(* IEC 61131-3 sources: beebread/doc (part 3) *)

FUNCTION OSCAT_VERSION : DWORD
VAR_INPUT
	IN : BOOL;
END_VAR

IF in THEN
	OSCAT_VERSION := DATE_TO_DWORD(D#2024-07-16);
ELSE
	OSCAT_VERSION := 335;
END_IF;
END_FUNCTION

FUNCTION STATUS_TO_ESR : esr_data
VAR_INPUT
	status : BYTE;
	adress : STRING(10);
	DT_in : DT;
	TS : TIME;
END_VAR

IF status < 100 THEN
	status_to_ESR.typ := 1;
ELSIF status < 200 THEN
	status_to_ESR.typ := 2;
ELSE
	status_to_ESR.typ := 3;
END_IF;
status_to_ESR.adress:= adress;
status_to_ESR.DS := DT_in;
status_to_ESR.TS := TS;
status_to_ESR.data[0] := status;
END_FUNCTION

// Commented out for beedance: it reads or writes the bytes of a STRING through a pointer; a beedance reference (REF_TO) refers to a whole variable of its type.
// FUNCTION BIN_TO_BYTE : BYTE
// VAR_INPUT
// 	BIN : STRING(12);
// END_VAR
// VAR
// 	pt : REF_TO BYTE;
// 	i: INT;
// 	X: BYTE;
// 	stop: INT;
// END_VAR
//
// pt := REF(bin);
// stop := LEN(bin);
// FOR I := 1 TO stop DO
// 	x := pt^;
// 	(* calculate the value of the digit *)
// 	IF X = 48 THEN
// 		BIN_TO_BYTE := SHL(BIN_TO_BYTE,1);
// 	ELSIF X = 49 THEN
// 		BIN_TO_BYTE := SHL(BIN_TO_BYTE,1) OR 1;
// 	END_IF;
// 	pt := pt + 1;
// END_FOR;
// END_FUNCTION

// Commented out for beedance: it reads or writes the bytes of a STRING through a pointer; a beedance reference (REF_TO) refers to a whole variable of its type.
// FUNCTION BIN_TO_DWORD : DWORD
// VAR_INPUT
// 	BIN : STRING(40);
// END_VAR
// VAR
// 	pt : REF_TO BYTE;
// 	i: INT;
// 	X: BYTE;
// 	stop: INT;
// END_VAR
//
// pt := REF(bin);
// stop := LEN(bin);
// FOR I := 1 TO stop DO
// 	x := pt^;
// 	(* calculate the value of the digit *)
// 	IF X = 48 THEN
// 		BIN_TO_DWORD := SHL(BIN_TO_DWORD,1);
// 	ELSIF X = 49 THEN
// 		BIN_TO_DWORD := SHL(BIN_TO_DWORD,1) OR 1;
// 	END_IF;
// 	pt := pt + 1;
// END_FOR;
// END_FUNCTION

// Commented out for beedance: it computes with pointers as addresses (pt := pt + 1); beedance references (REF_TO) have no arithmetic.
// FUNCTION BYTE_TO_STRB : STRING(8)
// VAR_INPUT
// 	IN : BYTE;
// END_VAR
// VAR
// 	i: INT;
// 	pt : REF_TO BYTE;
// END_VAR
//
// (* determine pointer for the output *)
// pt := REF(BYTE_TO_STRB);
// (* determine and write the 8 output characters *)
// FOR i := 1 TO 8 DO
// 	pt^ := BOOL_TO_BYTE(in.7) + 48;
// 	in := SHL(in,1);
// 	pt := pt + 1;
// END_FOR;
//
// (* the output string still has to be terminated with 0 *)
// pt^ := 0;
// END_FUNCTION

// Commented out for beedance: it computes with pointers as addresses (pt := pt + 1); beedance references (REF_TO) have no arithmetic.
// FUNCTION BYTE_TO_STRH : STRING(2)
// VAR_INPUT
// 	IN : BYTE;
// END_VAR
// VAR
// 	temp : BYTE;
// 	PT : REF_TO BYTE;
// END_VAR
//
// (* read pointer to output string *)
// PT := REF(BYTE_TO_STRH);
// (* calculate high order hex value *)
// temp := SHR(in,4);
// (* convert value to hex character *)
// IF temp <= 9 THEN temp := temp + 48; ELSE temp := temp + 55; END_IF;
// (* write friat character to output string *)
// PT^ := temp;
// (* calculate low order hex value *)
// temp := in AND 2#00001111;
// IF temp <= 9 THEN temp := temp + 48; ELSE temp := temp + 55; END_IF;
// (* increment pointer and wirte low order character *)
// pt := pt + 1;
// pt^ := temp;
// (* set pointer at the end of the output string and close the string with 0 *)
// pt := pt + 1;
// pt^:= 0;
// END_FUNCTION

// Commented out for beedance: it computes with pointers as addresses (pt := pt + 1); beedance references (REF_TO) have no arithmetic.
// FUNCTION CAPITALIZE : STRING(STRING_LENGTH)
// VAR_INPUT
// 	str : STRING(STRING_LENGTH);
// END_VAR
// VAR
// 	PT : REF_TO BYTE;
// 	pos : INT;
// 	L : INT;
// 	first : BOOL := TRUE;
// END_VAR
//
// PT := REF(CAPITALIZE);
// CAPITALIZE := str;
// L := LEN(str);
// FOR pos := 1 TO l DO
// 	IF first THEN pt^ := TO_UPPER(pt^);	END_IF;
// 	(* remember in first if the next char needs to capitalized *)
// 	first := pt^= 32;
// 	PT := pt + 1;
// END_FOR;
// END_FUNCTION

// Commented out for beedance: it uses CODE, which is commented out.
// FUNCTION CHARCODE : BYTE
// VAR_INPUT
// 	STR : STRING(10);
// END_VAR
// VAR
// 	found: STRING(1);
// 	search : STRING(10);
// 	pos: INT;
// 	i: INT;
// END_VAR
//
// IF LEN(str) = 1 THEN
// 	CHARCODE := CODE(STR, 1);
// ELSIF str <> '' THEN
// 	(* construct search string *)
// 	search := CONCAT('&', str);
// 	search := CONCAT(search, ';');
// 	WHILE pos = 0 AND (i < 4) DO
// 		i := i + 1;
// 		pos := FIND(setup.CHARNAMES[i], search);
// 	END_WHILE;
// 	found := MID(setup.CHARNAMES[i], 1, pos - 1);
// 	CHARCODE := CODE(found, 1);
// END_IF;
// END_FUNCTION

// Commented out for beedance: it uses CHR_TO_STRING, which is commented out.
// FUNCTION CHARNAME : STRING(10)
// VAR_INPUT
// 	C : BYTE;
// END_VAR
// VAR
// 	pos: INT;
// 	i : INT;
// END_VAR
//
// IF C <> 0 THEN
// 	(* construct search string from code followed by $ sign, also clear charname string*)
// 	CHARNAME := CHR_TO_STRING(C);
// 	CHARNAME := CONCAT(CHARNAME,'&');
// 	CHARNAME := CONCAT(';', CHARNAME);
// 	WHILE pos = 0 AND (i < 4) DO
// 		i := i + 1;
// 		pos := FIND(setup.CHARNAMES[i], CHARNAME);
// 	END_WHILE;
// 	IF pos > 0 THEN
// 		CHARNAME := MID(setup.CHARNAMES[i], 10, pos + 3);
// 		(* search for end of name and truncate *)
// 		pos := FIND(CHARNAME, ';');
// 		CHARNAME := LEFT(CHARNAME,pos - 1);
// 	ELSE
// 		CHARNAME := CHR_TO_STRING(C);
// 	END_IF;
// ELSE
// 	CHARNAME := '';
// END_IF;
// END_FUNCTION

// Commented out for beedance: it computes with pointers as addresses (pt := pt + 1); beedance references (REF_TO) have no arithmetic.
// FUNCTION CHR_TO_STRING : STRING(1)
// VAR_INPUT
// 	C : BYTE;
// END_VAR
// VAR
// 	PT : REF_TO BYTE;
// END_VAR
//
// PT := REF(CHR_TO_STRING);
// PT^ := C;
// pt := pt + 1;
// pt^ := 0;
// END_FUNCTION

FUNCTION CLEAN : STRING(STRING_LENGTH)
VAR_INPUT
	IN : STRING(STRING_LENGTH);
	CX : STRING(80);
END_VAR
VAR
	pos: INT := 1;
	stop: INT;
END_VAR

(* copy input string *)
CLEAN := IN;
stop := LEN(in);
WHILE pos <= stop DO
	IF FIND(cx, MID(CLEAN, 1, pos)) > 0 THEN
		(* charcter found skip to next one *)
		pos := pos + 1;
	ELSE
		(* wrong chracter needs to be deleted *)
		CLEAN := DELETE(CLEAN, 1, pos);
		stop := stop - 1;	(* the string is one character shorter now *)
	END_IF;
END_WHILE;
END_FUNCTION

// Commented out for beedance: it computes with pointers as addresses (pt := pt + 1); beedance references (REF_TO) have no arithmetic.
// FUNCTION CODE : BYTE
// VAR_INPUT
// 	STR : STRING(STRING_LENGTH);
// 	POS : INT;
// END_VAR
// VAR
// 	PT : REF_TO BYTE;
// END_VAR
//
// IF pos < 1 OR pos > LEN(str) THEN
// 	CODE := 0;
// 	RETURN;
// ELSE
// 	PT := REF(STR) + INT_TO_DWORD(pos - 1);
// 	CODE := pt^;
// END_IF;
// END_FUNCTION

// Commented out for beedance: it reads or writes the bytes of a STRING through a pointer; a beedance reference (REF_TO) refers to a whole variable of its type.
// FUNCTION COUNT_CHAR : INT
// VAR_INPUT
// 	str : STRING(STRING_LENGTH);
// 	chr : BYTE;
// END_VAR
// VAR
// 	l: INT;
// 	pt : REF_TO BYTE;
// 	pos: INT;
// END_VAR
//
// PT := REF(str);
// l := LEN(str);
// COUNT_CHAR := 0;
// FOR pos := 1 TO l DO
// 	IF pt^ = CHR THEN COUNT_CHAR := COUNT_CHAR + 1; END_IF;
//     PT := PT + 1;
// END_FOR;
// END_FUNCTION

FUNCTION COUNT_SUBSTRING : INT
VAR_INPUT
   SEARCH : STRING;
   STR : STRING;
END_VAR
VAR
   pos : INT;
   size : INT;
END_VAR
VAR
	STR_work : STRING;
END_VAR
(* IEC 61131-3 does not let a POU assign to its inputs, so the body works on copies. *)
STR_work := STR;

COUNT_SUBSTRING := 0;
size := LEN(SEARCH);
REPEAT
   pos := FIND(STR_work,SEARCH);
   IF pos > 0 THEN
      STR_work := REPLACE(STR_work, '', size,pos);
      COUNT_SUBSTRING := COUNT_SUBSTRING + 1;
   END_IF;
UNTIL pos = 0
END_REPEAT;
END_FUNCTION

// Commented out for beedance: it reads or writes the bytes of a STRING through a pointer; a beedance reference (REF_TO) refers to a whole variable of its type.
// FUNCTION DEC_TO_BYTE : BYTE
// VAR_INPUT
// 	DEC : STRING(10);
// END_VAR
// VAR
// 	pt : REF_TO BYTE;
// 	i: INT;
// 	X: BYTE;
// 	stop: INT;
// END_VAR
//
// pt := REF(dec);
// stop := LEN(DEC);
// FOR I := 1 TO stop DO
// 	(* read the first character and subtract 48 to get value in decimal 0 = 48 *)
// 	x := pt^;
// 	(* calculate the value of the digit *)
// 	IF X > 47 AND x < 58 THEN
// 		DEC_TO_BYTE := DEC_TO_BYTE * 10 + X - 48;
// 	END_IF;
// 	pt := pt + 1;
// END_FOR;
// END_FUNCTION

// Commented out for beedance: it reads or writes the bytes of a STRING through a pointer; a beedance reference (REF_TO) refers to a whole variable of its type.
// FUNCTION DEC_TO_DWORD : DWORD
// VAR_INPUT
// 	DEC : STRING(20);
// END_VAR
// VAR
// 	pt : REF_TO BYTE;
// 	i: INT;
// 	X: BYTE;
// 	stop: INT;
// END_VAR
//
// pt := REF(dec);
// stop := LEN(dec);
// FOR I := 1 TO stop DO
// 	(* read the first character and subtract 48 to get value in decimal 0 = 48 *)
// 	x := pt^;
// 	(* calculate the value of the digit *)
// 	IF X > 47 AND x < 58 THEN
// 		DEC_TO_DWORD := DEC_TO_DWORD * 10 + X - 48;
// 	END_IF;
// 	pt := pt + 1;
// END_FOR;
// END_FUNCTION

// Commented out for beedance: it reads or writes the bytes of a STRING through a pointer; a beedance reference (REF_TO) refers to a whole variable of its type.
// FUNCTION DEC_TO_INT : INT
// VAR_INPUT
// 	DEC : STRING(10);
// END_VAR
// VAR
// 	pt : REF_TO BYTE;
// 	i: INT;
// 	X: BYTE;
// 	sign: BOOL;
// 	stop: INT;
// END_VAR
//
// pt := REF(dec);
// stop := LEN(dec);
// FOR I := 1 TO stop DO
// 	(* read the first character and subtract 48 to get value in decimal 0 = 48 *)
// 	x := pt^;
// 	(* calculate the value of the digit *)
// 	IF X > 47 AND x < 58 THEN
// 		DEC_TO_INT := DEC_TO_INT * 10 + X - 48;
// 	ELSIF X = 45 AND DEC_TO_INT = 0 THEN
// 		sign := TRUE;
// 	END_IF;
// 	pt := pt + 1;
// END_FOR;
// IF sign THEN DEC_TO_INT := -DEC_TO_INT; END_IF;
// END_FUNCTION

FUNCTION DEL_CHARS : STRING(STRING_LENGTH)
VAR_INPUT
	IN : STRING(STRING_LENGTH);
	CX : STRING(80);
END_VAR
VAR
	pos: INT := 1;
	stop: INT;
END_VAR

(* copy input string *)
DEL_CHARS := IN;
stop := LEN(in);
WHILE pos <= stop DO
	IF FIND(cx, MID(DEL_CHARS, 1, pos)) > 0 THEN
		(* wrong chracter needs to be deleted *)
		DEL_CHARS := DELETE(DEL_CHARS, 1, pos);
		stop := stop - 1;	(* the string is one character shorter now *)
	ELSE
		(* charcter not found skip to next one *)
		pos := pos + 1;
	END_IF;
END_WHILE;
END_FUNCTION

// Commented out for beedance: it uses CODE, which is commented out.
// FUNCTION DT_TO_STRF : STRING
// VAR_INPUT
// 	DTI : DT;
// 	MS : INT;
// 	FMT : STRING;
// 	LANG : INT;
// END_VAR
// VAR CONSTANT
// 	FILL : STRING(1) := '0';
// 	BLANK : STRING(1) := ' ';
// END_VAR
// VAR
// 	ly : INT;
// 	dx: DATE;
// 	fs: STRING(10);
// 	td: TOD;
// 	tmp : INT;
// 	pos : INT;
// 	f : INT;
// END_VAR
//
// IF LANG < 1 THEN ly := language.DEFAULT; ELSE ly := MIN(language.LMAX, LANG); END_IF;
//
// (* decode date and time information *)
// dx := DT_TO_DATE(DTI);
// td := DT_TO_TOD(DTI);
//
// (* parse the format string *)
// DT_TO_STRF := FMT;
// pos := FIND(DT_TO_STRF, '#');
// WHILE pos > 0 DO
// 	(* retrieve format identifier *)
// 	f := CODE(DT_TO_STRF, pos + 1);
// 	(* generate the return string according to the format character *)
// 	fs := '';
// 	CASE f OF
// 		65 : (* letter A retunrs the year in 4 digits *)
// 			fs := INT_TO_STRING(YEAR_OF_DATE(dx));
// 		66 : (* letter B returns the year in exactly 2 digits *)
// 			fs := RIGHT(INT_TO_STRING(YEAR_OF_DATE(dx)),2);
// 		67 : (* letter C returns the month with 1 or 2 digits *)
// 			fs := INT_TO_STRING(MONTH_OF_DATE(dx));
// 		68 : (* letter D returns the month with exactly 2 digits *)
// 			fs := INT_TO_STRING(MONTH_OF_DATE(dx));
// 			IF LEN(fs) < 2 THEN fs := CONCAT('0', fs); END_IF;
// 		69 : (* letter E returns the month with 3 characters *)
// 			fs := MONTH_TO_STRING(MONTH_OF_DATE(dx), ly, 3);
// 		70 : (* letter F returns the month with all characters *)
// 			fs := MONTH_TO_STRING(MONTH_OF_DATE(dx), ly, 0);
// 		71 : (* letter G returns the day with up to 2 digits *)
// 			fs := INT_TO_STRING(DAY_OF_MONTH(dx));
// 		72 : (* letter H returns the day of the month with exactly 2 digits *)
// 			fs := INT_TO_STRING(DAY_OF_MONTH(dx));
// 			IF LEN(fs) < 2 THEN fs := CONCAT(FILL, fs); END_IF;
// 		73 : (* letter I returns the weekday as the number 1..7 1 = monday *)
// 			fs := INT_TO_STRING(DAY_OF_WEEK(dx));
// 		74 : (* letter J returns the weekday in 2 character writing *)
// 			fs := WEEKDAY_TO_STRING(DAY_OF_WEEK(dx), ly, 2);
// 		75 : (* letter K returns the weekday with all characters *)
// 			fs := WEEKDAY_TO_STRING(DAY_OF_WEEK(dx), ly, 0);
// 		76 : (* letter L returns AM or PM for the given DateTime *)
// 			IF td >= TOD#12:00:00 THEN fs := 'PM'; ELSE fs := 'AM'; END_IF;
// 		77 : (* letter M returns the hour in 1 or 2 digit form 0..24h *)
// 			fs := INT_TO_STRING(HOUR(td));
// 		78 : (* letter N returns the hour in exactly 2 digit form 0..24h *)
// 			fs := INT_TO_STRING(HOUR(td));
// 			IF LEN(fs) < 2 THEN fs := CONCAT(FILL, fs); END_IF;
// 		79 : (* letter O returns the hour in 1 or 2 digit form 0..12h *)
// 			tmp := HOUR(td) MOD 12;
// 			IF tmp = 0 THEN tmp := 12; END_IF;
// 			fs := INT_TO_STRING(tmp);
// 		80 : (* letter P returns the hour in exactly 2 digit form 0..12h *)
// 			tmp := HOUR(td) MOD 12;
// 			IF tmp = 0 THEN tmp := 12; END_IF;
// 			fs := INT_TO_STRING(tmp);
// 			IF LEN(fs) < 2 THEN fs := CONCAT(FILL, fs); END_IF;
// 		81 : (* letter Q returns the minute of the hour in 1 or two digit form *)
// 			fs := INT_TO_STRING(MINUTE(td));
// 		82 : (* letter R returns the minute of the hour in exactly two digit form *)
// 			fs := INT_TO_STRING(MINUTE(td));
// 			IF LEN(fs) < 2 THEN fs := CONCAT(FILL, fs); END_IF;
// 		83 : (* letter S returns the second of the minute in 1 or two digit form *)
// 			fs := INT_TO_STRING(REAL_TO_INT(SECOND(td)));
// 		84 : (* letter T returns the second of the minute in exactly two digit form *)
// 			fs := INT_TO_STRING(REAL_TO_INT(SECOND(td)));
// 			IF LEN(fs) < 2 THEN fs := CONCAT(FILL, fs); END_IF;
// 		85 : (* letter U returns the milliseconds in 1 to 3 digits *)
// 			fs := INT_TO_STRING(MS);
// 		86 : (* letter V returns the milliseconds in exactly 3 digit form *)
// 			fs := INT_TO_STRING(MS);
// 			fs := CONCAT('00',fs);
// 			fs := RIGHT(fs, 3);
// 		87 : (* letter W returns the day of the month with exactly 2 digits first digit is filled with blank if necessary *)
// 			fs := INT_TO_STRING(DAY_OF_MONTH(dx));
// 			IF LEN(fs) < 2 THEN fs := CONCAT(BLANK, fs); END_IF;
// 		88 : (* letter X returns the month with exactly 2 digits first digit is filled with blank if necessary *)
// 			fs := INT_TO_STRING(MONTH_OF_DATE(dx));
// 			IF LEN(fs) < 2 THEN fs := CONCAT(BLANK, fs); END_IF;
// 		END_CASE;
// 	DT_TO_STRF := REPLACE(DT_TO_STRF, fs, 2, pos);
// 	pos := FIND(DT_TO_STRF, '#');
// END_WHILE;
// END_FUNCTION

// Commented out for beedance: it computes with pointers as addresses (pt := pt + 1); beedance references (REF_TO) have no arithmetic.
// FUNCTION DWORD_TO_STRB : STRING(32)
// VAR_INPUT
// 	IN : DWORD;
// END_VAR
// VAR
// 	pt : REF_TO BYTE;
// 	i: INT;
// END_VAR
//
// (* determine pointer for the output *)
// pt := REF(DWORD_TO_STRB);
// (* determine and write the 8 output characters *)
// FOR i := 1 TO 32 DO
// 	pt^:= BOOL_TO_BYTE(in.31) + 48;
// 	in := SHL(in,1);
// 	pt := pt + 1;
// END_FOR;
//
// (* the output string still has to be terminated with 0 *)
// pt^ := 0;
// END_FUNCTION

// Commented out for beedance: it uses FIX, which is commented out.
// FUNCTION DWORD_TO_STRF : STRING(20)
// VAR_INPUT
// 	IN : DWORD;
// 	N : INT;
// END_VAR
//
// (* limit N to max 20 characters *)
// (* convert dword to string first and cut to length N *)
// DWORD_TO_STRF := FIX(DWORD_TO_STRING(in),LIMIT(0,N,20),48,1);
// END_FUNCTION

// Commented out for beedance: it computes with pointers as addresses (pt := pt + 1); beedance references (REF_TO) have no arithmetic.
// FUNCTION DWORD_TO_STRH : STRING(8)
// VAR_INPUT
// 	IN : DWORD;
// END_VAR
// VAR
// 	i : INT;
// 	temp : BYTE;
// 	pt : REF_TO BYTE;
// END_VAR
//
// (* read output adress to pointer *)
// pt := REF(DWORD_TO_STRH) + 8;
// (* wirte the closing byte for the string *)
// pt^:= 0;
//
// (* write the 8 hex characters backwards *)
// FOR i := 1 TO 8 DO;
// 	(* decrement the pointer *)
// 	pt := pt - 1;
// 	(* read the lowest order hex value *)
// 	temp := DWORD_TO_BYTE(in AND 16#0000000F);
// 	(* convert value to hex character *)
// 	IF temp <= 9 THEN temp := temp + 48; ELSE temp := temp + 55; END_IF;
// 	(* write character to output string *)
// 	PT^ := temp;
// 	(* shift in for nect hex character *)
// 	in := SHR(in,4);
// END_FOR;
// END_FUNCTION

// Commented out for beedance: it uses UPPERCASE, which is commented out.
// FUNCTION EXEC : STRING(STRING_LENGTH)
// VAR_INPUT
// 	str : STRING(STRING_LENGTH);
// END_VAR
// VAR
// 	pos: INT;
// 	R1: REAL;
// 	R2: REAL;
// 	operator: STRING(10);
// END_VAR
//
// (* extract both numbers and operator *)
// EXEC := UPPERCASE(TRIM(str));
//
// pos := FINDB_NONUM(EXEC);
// IF pos > 1 THEN R1 := STRING_TO_REAL(LEFT(EXEC,pos-1)); END_IF;
// R2 := STRING_TO_REAL(RIGHT(EXEC,LEN(EXEC)-pos));
// EXEC := LEFT(EXEC,pos);
// pos := FINDB_NUM(EXEC);
// operator := RIGHT(EXEC,LEN(EXEC) - pos);
// IF operator = '' AND LEN(str) = 0 THEN
// 	EXEC := '';
// 	RETURN;
// ELSIF operator = '' THEN
// 	EXEC := str;
// 	RETURN;
// END_IF;
// IF operator = '^' THEN
// 	EXEC := REAL_TO_STRING(EXPT(R1, R2));
// ELSIF operator = 'SQRT' THEN
// 	EXEC := REAL_TO_STRING(SQRT(R2));
// ELSIF operator = 'SIN' THEN
// 	EXEC := REAL_TO_STRING(SIN(r2));
// ELSIF operator = 'COS' THEN
// 	EXEC := REAL_TO_STRING(COS(r2));
// ELSIF operator = 'TAN' THEN
// 	EXEC := REAL_TO_STRING(TAN(R2));
// ELSIF operator = '*' THEN
// 	EXEC := REAL_TO_STRING(R1 * R2);
// ELSIF operator = '/' THEN
// 	IF R2 <> 0 THEN EXEC := REAL_TO_STRING(R1 / R2); ELSE EXEC := 'ERROR'; END_IF;
// ELSIF operator = '+' THEN
// 	EXEC := REAL_TO_STRING(r1 + r2);
// ELSIF operator = '-' THEN
// 	EXEC := REAL_TO_STRING(r1 - r2);
// ELSE
// 	EXEC := 'ERROR';
// END_IF;
//
// IF EXEC = 'ERROR' THEN
// 	RETURN;
// (* some systems deliver integer instead of real *)
// ELSIF FIND(EXEC,'.') = 0 THEN
// 	EXEC := CONCAT(EXEC, '.0');
// (* some systems deliver n. instead of n.0 ! *)
// ELSIF RIGHT(EXEC,1) = '.' THEN
// 	EXEC := CONCAT(EXEC,'0');
// END_IF;
// END_FUNCTION

// Commented out for beedance: it uses CHR_TO_STRING, which is commented out.
// FUNCTION FILL : STRING(STRING_LENGTH)
// VAR_INPUT
// 	C : BYTE;
// 	L : INT;
// END_VAR
// VAR
// 	i: INT;
// 	sx: STRING(1);
// END_VAR
// VAR
// 	L_work : INT;
// END_VAR
// (* IEC 61131-3 does not let a POU assign to its inputs, so the body works on copies. *)
// L_work := L;
//
// Sx := CHR_TO_STRING(c);
// (* limit L to maximum 80 characters the length of a standard string *)
// L_work := LIMIT(0,L_work,STRING_LENGTH);
// (* create a string of characters to be connected to str *)
// FOR i := 1 TO 8 DO
// 	FILL := CONCAT(FILL,FILL);
// 	IF L_work.7 THEN FILL := CONCAT(FILL,Sx); END_IF;
// 	L_work := SHL(L_work,1);
// END_FOR;
// END_FUNCTION

// Commented out for beedance: it reads or writes the bytes of a STRING through a pointer; a beedance reference (REF_TO) refers to a whole variable of its type.
// FUNCTION FIND_CHAR : INT
// VAR_INPUT
// 	str : STRING(STRING_LENGTH);
// 	pos : INT;
// END_VAR
// VAR
// 	i: INT;
// 	pt : REF_TO ARRAY[1..255] OF BYTE;
// 	stop: INT;
// 	X: BYTE;
// END_VAR
//
// pt := REF(str);
// stop := LEN(str);
// FOR i := MAX(pos,1) TO stop DO;
// 	X := pt^[i];
// 	IF X > 31 AND ((setup.EXTENDED_ASCII AND X <> 127) OR (NOT setup.EXTENDED_ASCII AND X < 127)) THEN
// 		FIND_CHAR := i;
// 		RETURN;
// 	END_IF;
// END_FOR;
// FIND_CHAR := 0;
// END_FUNCTION

// Commented out for beedance: it reads or writes the bytes of a STRING through a pointer; a beedance reference (REF_TO) refers to a whole variable of its type.
// FUNCTION FIND_CTRL : INT
// VAR_INPUT
// 	str : STRING(STRING_LENGTH);
// 	pos : INT;
// END_VAR
// VAR
// 	i: INT;
// 	pt : REF_TO ARRAY[1..255] OF BYTE;
// 	stop: INT;
// 	x: BYTE;
// END_VAR
//
// pt := REF(str);
// stop := LEN(str);
// FOR i := MAX(pos,1) TO stop DO;
// 	x := PT^[I];
// 	IF x < 32 OR X = 127 THEN
// 		FIND_CTRL := i;
// 		RETURN;
// 	END_IF;
// END_FOR;
// FIND_CTRL := 0;
// END_FUNCTION

// Commented out for beedance: it reads or writes the bytes of a STRING through a pointer; a beedance reference (REF_TO) refers to a whole variable of its type.
// FUNCTION FIND_NONUM : INT
// VAR_INPUT
// 	str : STRING(STRING_LENGTH);
// 	pos : INT;
// END_VAR
// VAR
// 	i: INT;
// 	pt : REF_TO ARRAY[1..255] OF BYTE;
// 	end: INT;
// 	X: BYTE;
// END_VAR
//
// pt := REF(str);
// end := LEN(str);
// FOR i := MAX(pos,1) TO end DO;
// 	X := pt^[i];
// 	IF (X < 48 AND X <> 46) OR X > 57 THEN
// 		FIND_NONUM := i;
// 		RETURN;
// 	END_IF;
// END_FOR;
// FIND_NONUM := 0;
// END_FUNCTION

// Commented out for beedance: it reads or writes the bytes of a STRING through a pointer; a beedance reference (REF_TO) refers to a whole variable of its type.
// FUNCTION FIND_NUM : INT
// VAR_INPUT
// 	str : STRING(STRING_LENGTH);
// 	pos : INT;
// END_VAR
// VAR
// 	i : INT;
// 	pt : REF_TO ARRAY[1..255] OF BYTE;
// 	stop : INT;
// 	X: BYTE;
// END_VAR
//
// pt := REF(str);
// stop := LEN(str);
// FOR i := MAX(pos,1) TO stop DO;
// 	X := pt^[i];
// 	IF (X > 47 AND X < 58) OR X = 46 THEN
// 		FIND_NUM := i;
// 		RETURN;
// 	END_IF;
// END_FOR;
// FIND_NUM := 0;
// END_FUNCTION

FUNCTION FINDB : INT
VAR_INPUT
	str1 : STRING(STRING_LENGTH);
	str2 : STRING(STRING_LENGTH);
END_VAR
VAR
	pos: INT;
	length: INT;
END_VAR

length := LEN(str2);
FOR pos := LEN(str1) - length + 1 TO 1 BY -1 DO
	IF MID(str1,length,pos) = str2 THEN
		FindB := pos;
		RETURN;
	END_IF;
END_FOR;
FindB := 0;
END_FUNCTION

// Commented out for beedance: it computes with pointers as addresses (pt := pt + 1); beedance references (REF_TO) have no arithmetic.
// FUNCTION FINDB_NONUM : INT
// VAR_INPUT
// 	str : STRING(STRING_LENGTH);
// END_VAR
// VAR
// 	pos: INT;
// 	pt : REF_TO BYTE;
// END_VAR
//
// pt := REF(str) + LEN(str) - 1;
// FOR pos := LEN(str) TO 1 BY -1 DO;
// 	IF (PT^ < 48 AND PT^ <> 46) OR PT^ > 57 THEN
// 		FINDB_NONUM := pos;
// 		RETURN;
// 	END_IF;
// 	PT := PT - 1;
// END_FOR;
// FINDB_NONUM := 0;
// END_FUNCTION

// Commented out for beedance: it computes with pointers as addresses (pt := pt + 1); beedance references (REF_TO) have no arithmetic.
// FUNCTION FINDB_NUM : INT
// VAR_INPUT
// 	str : STRING(STRING_LENGTH);
// END_VAR
// VAR
// 	pos: INT;
// 	pt : REF_TO BYTE;
// END_VAR
//
// pt := REF(str) + LEN(str) - 1;
// FOR pos := LEN(str) TO 1 BY -1 DO;
// 	IF (PT^ > 47 AND PT^ < 58) OR PT^ = 46 THEN
// 		FINDB_NUM := pos;
// 		RETURN;
// 	END_IF;
// 	PT := PT - 1;
// END_FOR;
// FINDB_NUM := 0;
// END_FUNCTION

FUNCTION FINDP : INT
VAR_INPUT
	str : STRING(STRING_LENGTH);
	src : STRING(STRING_LENGTH);
	pos: INT;
END_VAR
VAR
	i: INT;
	ls: INT;
	lx: INT;
	stp: INT;
END_VAR

ls := LEN(str);
lx := LEN(src);
IF ls < lx OR lx = 0 THEN RETURN; END_IF;
stp := ls - lx + 1;
FOR i := MAX(pos,1) TO stp DO
	IF MID(str,lx,i) = src THEN
		FINDP := i;
		RETURN;
	END_IF;
END_FOR;
FINDP := 0;
END_FUNCTION

// Commented out for beedance: it uses FILL, which is commented out.
// FUNCTION FIX : STRING(STRING_LENGTH)
// VAR_INPUT
// 	str : STRING(STRING_LENGTH);
// 	L : INT;
// 	C : BYTE;
// 	M : INT;
// END_VAR
// VAR
// 	N : INT;
// 	SX: STRING(STRING_LENGTH);
// END_VAR
//
// (* make sure L does not exceed the limits of a string *)
// N := LIMIT(0,L,STRING_LENGTH) - LEN(str);
// IF N <= 0 THEN
// 	(* truncate the string at length N *)
// 	IF M = 1 THEN
// 		FIX := RIGHT(str,L);
// 	ELSE
// 		FIX := LEFT(str,L);
// 	END_IF;
// ELSIF M = 1 THEN
// 	(* connect fill characters at the beginning *)
// 	sx := FILL(C,N);
// 	FIX := CONCAT(sx,str);
// ELSIF M = 2 THEN
// 	(* center str beween fill characters *)
// 	(* for an uneven number of fill characters, there is one more at the end *)
// 	sx := FILL(C,SHR(N+1,1));
// 	FIX := CONCAT(str,sx);
// 	SX := LEFT(sx,SHR(N,1));
// 	FIX := CONCAT(sx,FIX);
// ELSE
// 	(* connect fill characters at the end *)
// 	SX := FILL(C,N);
// 	FIX := CONCAT(str,SX);
// END_IF;
// END_FUNCTION

// Commented out for beedance: it reads or writes the bytes of a STRING through a pointer; a beedance reference (REF_TO) refers to a whole variable of its type.
// FUNCTION FLOAT_TO_REAL : REAL
// VAR_INPUT
// 	FLT : STRING(20);
// END_VAR
// VAR
// 	pt : REF_TO ARRAY[1..20] OF BYTE;
// 	i: INT;
// 	X: BYTE;
// 	sign: INT := 1;
// 	stop: INT;
// 	tmp: DINT;
// 	d : INT;
// END_VAR
//
// pt := REF(FLT);
// stop := LEN(FLT);
//
// (* we first check for sign and exit if first number or dot is reached *)
// FOR i := 1 TO stop DO
// 	X := pt^[i];
// 	IF X > 47 AND X < 58 OR X = 46 THEN
// 		EXIT;
// 	ELSIF X = 45 THEN
// 		(* code 45 is sign *)
// 		sign := -1;
// 	END_IF;
// END_FOR;
//
// (* now we scan numbers till end or dot or E is reached *)
// FOR i := i TO stop DO
// 	X := pt^[i];
// 	IF X = 44 OR X = 46 OR X = 69 OR X = 101 THEN
// 		EXIT;
// 	(* calculate the value of the digit *)
// 	ELSIF X > 47 AND x < 58 THEN
// 		tmp := tmp * 10 + X - 48;
// 	END_IF;
// END_FOR;
//
// (* process the portion after the comma if comma or dot is reached exit if exponent starts *)
// IF x = 44 OR X = 46 THEN
// 	FOR i := i + 1 TO stop DO
// 		X := pt^[i];
// 		IF X = 69 OR X = 101 THEN
// 			EXIT;
// 		ELSIF x > 47 AND x < 58 THEN
// 			tmp := tmp * 10 + X - 48;
// 			d := d - 1;
// 		END_IF;
// 	END_FOR;
// END_IF;
//
// (* process exponent if present *)
// IF X = 69 OR X = 101 THEN
// 	d := d + DEC_TO_INT(RIGHT(FLT, stop - i));
// END_IF;
//
// FLOAT_TO_REAL :=  EXPN(10, d) * DINT_TO_REAL(TMP * SIGN);
// END_FUNCTION

// Commented out for beedance: it uses BIN_TO_BYTE, which is commented out.
// FUNCTION FSTRING_TO_BYTE : BYTE
// VAR_INPUT
// 	IN : STRING(12);
// END_VAR
//
// IF LEFT(IN, 2) = '2#' THEN
// 	(* we need to convert binary *)
// 	FSTRING_TO_BYTE := BIN_TO_BYTE(RIGHT(in, LEN(in) - 2));
// ELSIF LEFT(in, 2) = '8#' THEN
// 	(* weneed to convert octals *)
// 	FSTRING_TO_BYTE := OCT_TO_BYTE(RIGHT(in, LEN(in) - 2));
// ELSIF LEFT(in, 3) = '16#' THEN
// 	(* we need to convert hexadecimal *)
// 	FSTRING_TO_BYTE := HEX_TO_BYTE(RIGHT(in, LEN(in) - 3));
// ELSE
// 	(* we assume decimal representation *)
// 	FSTRING_TO_BYTE := DEC_TO_BYTE(CLEAN(in,'0123456789'));
// END_IF;
// END_FUNCTION

// Commented out for beedance: it uses FSTRING_TO_MONTH, which is commented out.
// FUNCTION FSTRING_TO_DT : DT
// VAR_INPUT
// 	SDT : STRING(60);
// 	FMT : STRING(60);
// END_VAR
// VAR CONSTANT
// 	ignore: STRING(1) := '*';  (* ignore character is * *)
// 	fchar : STRING(1) := '#';  (* format character is # *)
// END_VAR
// VAR
// 	c: STRING(1);
// 	tmp: STRING(20);
// 	end: INT;
// 	dy : INT := 1970;
// 	dm : INT := 1;
// 	dd : INT := 1;
// 	th : INT;
// 	tm : INT;
// 	ts : INT;
// END_VAR
// VAR
// 	SDT_work : STRING;
// 	FMT_work : STRING;
// END_VAR
// (* IEC 61131-3 does not let a POU assign to its inputs, so the body works on copies. *)
// SDT_work := SDT;
// FMT_work := FMT;
//
// (* scan input string *)
// WHILE FMT_work <> '' DO
// 	c := LEFT(FMT_work,1);
// 	IF c = ignore THEN
// 		(* skip ignore characters *)
// 		FMT_work := DELETE(FMT_work,1,1);
// 		SDT_work := DELETE(SDT_work,1,1);
// 	ELSIF C = fchar THEN
// 		(* format chracter found skip format char and read identifier *)
// 		(* store format identifier in c and skip to next char in fmt *)
// 		c := MID(FMT_work,1,2);
// 		FMT_work := DELETE(FMT_work,2,1);
// 		(* extract the substring until the end of sdt or to next char of fmt *)
// 		IF FMT_work = '' THEN
// 			tmp := SDT_work;
// 		ELSE
// 			(* serach for end of substring *)
// 			end := FIND(SDT_work, LEFT(FMT_work,1))-1;
// 			tmp := LEFT(SDT_work, end);
// 			SDT_work := DELETE(SDT_work, end,1);
// 		END_IF;
// 		(* extract information from substring *)
// 		IF c = 'Y' THEN
// 			dy := STRING_TO_INT(tmp);
// 			IF dy < 100 THEN dy := dy + 2000; END_IF;
// 		ELSIF c = 'M' THEN
// 			dm := STRING_TO_INT(tmp);
// 		ELSIF c = 'N' THEN
// 			dm := FSTRING_TO_MONTH(tmp,0);
// 		ELSIF c = 'D' THEN
// 			dd := STRING_TO_INT(tmp);
// 		ELSIF c = 'h' THEN
// 			th := STRING_TO_INT(tmp);
// 		ELSIF c = 'm' THEN
// 			tm := STRING_TO_INT(tmp);
// 		ELSIF c = 's' THEN
// 			ts := STRING_TO_INT(tmp);
// 		END_IF;
// 	ELSIF c = LEFT(SDT_work,1) THEN
// 		(* skip matching characters *)
// 		FMT_work := DELETE(FMT_work,1,1);
// 		SDT_work := DELETE(SDT_work,1,1);
// 	ELSE
// 		RETURN;
// 	END_IF;
// END_WHILE;
//
// FSTRING_TO_DT := SET_DT(dy,dm,dd,th,tm,ts);
// END_FUNCTION

// Commented out for beedance: it uses BIN_TO_DWORD, which is commented out.
// FUNCTION FSTRING_TO_DWORD : DWORD
// VAR_INPUT
// 	IN : STRING(40);
// END_VAR
//
// IF LEFT(IN, 2) = '2#' THEN
// 	(* we need to convert binary *)
// 	FSTRING_TO_DWORD := BIN_TO_DWORD(RIGHT(in, LEN(in) - 2));
// ELSIF LEFT(in, 2) = '8#' THEN
// 	(* weneed to convert octals *)
// 	FSTRING_TO_DWORD := OCT_TO_DWORD(RIGHT(in, LEN(in) - 2));
// ELSIF LEFT(in, 3) = '16#' THEN
// 	(* we need to convert hexadecimal *)
// 	FSTRING_TO_DWORD := HEX_TO_DWORD(RIGHT(in, LEN(in) - 3));
// ELSE
// 	(* we assume decimal representation *)
// 	FSTRING_TO_DWORD := DEC_TO_DWORD(CLEAN(in,'0123456789'));
// END_IF;
// END_FUNCTION

// Commented out for beedance: it uses CAPITALIZE, which is commented out.
// FUNCTION FSTRING_TO_MONTH : INT
// VAR_INPUT
// 	MTH : STRING(20);
// 	LANG : INT;
// END_VAR
// VAR
// 	lx: INT;
// END_VAR
// VAR
// 	MTH_work : STRING;
// END_VAR
// (* IEC 61131-3 does not let a POU assign to its inputs, so the body works on copies. *)
// MTH_work := MTH;
//
// IF LANG = 0 THEN lx := LANGUAGE.DEFAULT; ELSE lx := MIN(LANG, LANGUAGE.LMAX); END_IF;
// MTH_work := TRIM(MTH_work);
// MTH_work := CAPITALIZE(LOWERCASE(MTH_work));
//
// FOR FSTRING_TO_MONTH := 1 TO 12 DO
// 	IF MTH_work = language.MONTHS[lx, FSTRING_TO_MONTH] THEN RETURN; END_IF;
// 	IF MTH_work = language.MONTHS3[lx, FSTRING_TO_MONTH] THEN RETURN; END_IF;
// END_FOR;
//
// (* since no name matched try to decode as integer *)
// FSTRING_TO_MONTH := STRING_TO_INT(MTH_work);
// END_FUNCTION

// Commented out for beedance: it uses FSTRING_TO_WEEKDAY, which is commented out.
// FUNCTION FSTRING_TO_WEEK : BYTE
// VAR_INPUT
// 	WEEK : STRING(60);
// 	LANG : INT;
// END_VAR
// VAR
// 	pos: INT;
// END_VAR
// VAR
// 	WEEK_work : STRING;
// END_VAR
// (* IEC 61131-3 does not let a POU assign to its inputs, so the body works on copies. *)
// WEEK_work := WEEK;
//
// pos := FIND(WEEK_work, ',');
// WHILE pos > 0 DO
// 	FSTRING_TO_WEEK := FSTRING_TO_WEEK OR SHR(BYTE#128, FSTRING_TO_WEEKDAY(MID(WEEK_work, pos - 1, 1), LANG));
// 	WEEK_work := RIGHT(WEEK_work, LEN(WEEK_work) - pos);
// 	pos := FIND(WEEK_work, ',');
// END_WHILE;
// FSTRING_TO_WEEK := (FSTRING_TO_WEEK OR SHR(BYTE#128, FSTRING_TO_WEEKDAY(WEEK_work, LANG))) AND BYTE#127;
// END_FUNCTION

// Commented out for beedance: it uses CAPITALIZE, which is commented out.
// FUNCTION FSTRING_TO_WEEKDAY : INT
// VAR_INPUT
// 	WDAY : STRING(20);
// 	LANG : INT;
// END_VAR
// VAR
// 	tmp: STRING(2);
// 	i: INT;
// 	ly: INT;
// END_VAR
//
// IF LANG = 0 THEN ly := LANGUAGE.DEFAULT; ELSE ly := MIN(LANG, LANGUAGE.LMAX); END_IF;
// (* tmp needs to be calculated first otherwise find can return wrong values *)
// tmp := TRIM(wday);
// tmp := CAPITALIZE(LOWERCASE(tmp));
// FOR i := 1 TO 7 DO
// 	IF language.WEEKDAYS2[ly, i] = tmp THEN
// 		FSTRING_TO_WEEKDAY := i;
// 		RETURN;
// 	END_IF;
// END_FOR;
// FSTRING_TO_WEEKDAY := STRING_TO_INT(WDAY);
// END_FUNCTION

// Commented out for beedance: it reads or writes the bytes of a STRING through a pointer; a beedance reference (REF_TO) refers to a whole variable of its type.
// FUNCTION HEX_TO_BYTE : BYTE
// VAR_INPUT
// 	HEX : STRING(5);
// END_VAR
// VAR
// 	pt : REF_TO BYTE;
// 	i: INT;
// 	X: BYTE;
// 	stop: INT;
// END_VAR
//
// pt := REF(hex);
// stop := LEN(hex);
// FOR I := 1 TO stop DO
// 	(* read the first character and subtract 48 to get value in decimal 0 = 48 *)
// 	x := pt^;
// 	(* calculate the value of the digit *)
// 	IF X > 47 AND x < 58 THEN
// 		HEX_TO_BYTE := SHL(HEX_TO_BYTE,4) + X - 48;
// 	ELSIF X > 64 AND X < 71 THEN
// 		HEX_TO_BYTE := SHL(HEX_TO_BYTE,4) + X - 55;
// 	ELSIF X > 96 AND X < 103 THEN
// 		HEX_TO_BYTE := SHL(HEX_TO_BYTE,4) + X - 87;
// 	END_IF;
// 	pt := pt + 1;
// END_FOR;
// END_FUNCTION

// Commented out for beedance: it reads or writes the bytes of a STRING through a pointer; a beedance reference (REF_TO) refers to a whole variable of its type.
// FUNCTION HEX_TO_DWORD : DWORD
// VAR_INPUT
// 	Hex : STRING(20);
// END_VAR
// VAR
// 	pt : REF_TO BYTE;
// 	i: INT;
// 	X: BYTE;
// 	stop: INT;
// END_VAR
//
// pt := REF(hex);
// stop := LEN(hex);
// FOR I := 1 TO stop DO
// 	(* read the first character and subtract 48 to get value in decimal 0 = 48 *)
// 	x := pt^;
// 	(* calculate the value of the digit *)
// 	IF X > 47 AND x < 58 THEN
// 		HEX_TO_DWORD := SHL(HEX_TO_DWORD,4) + X - 48;
// 	ELSIF X > 64 AND X < 71 THEN
// 		HEX_TO_DWORD := SHL(HEX_TO_DWORD,4) + X - 55;
// 	ELSIF X > 96 AND X < 103 THEN
// 		HEX_TO_DWORD := SHL(HEX_TO_DWORD,4) + X - 87;
// 	END_IF;
// 	pt := pt + 1;
// END_FOR;
// END_FUNCTION

// Commented out for beedance: it reads or writes the bytes of a STRING through a pointer; a beedance reference (REF_TO) refers to a whole variable of its type.
// FUNCTION IS_ALNUM : BOOL
// VAR_INPUT
// 	str : STRING(STRING_LENGTH);
// END_VAR
// VAR
// 	L: INT;
// 	pt : REF_TO BYTE;
// 	pos: INT;
// END_VAR
//
// PT := REF(str);
// L := LEN(str);
// FOR pos := 1 TO L DO
// 	IF NOT (ISC_ALPHA(pt^) OR ISC_NUM(pt^)) THEN
// 		IS_ALNUM := FALSE;
// 		RETURN;
// 	END_IF;
//     	PT := PT + 1;
// END_FOR;
// IS_ALNUM := L > 0;
// END_FUNCTION

// Commented out for beedance: it reads or writes the bytes of a STRING through a pointer; a beedance reference (REF_TO) refers to a whole variable of its type.
// FUNCTION IS_ALPHA : BOOL
// VAR_INPUT
// 	str : STRING(STRING_LENGTH);
// END_VAR
// VAR
// 	L: INT;
// 	pt : REF_TO BYTE;
// 	pos: INT;
// END_VAR
//
// PT := REF(str);
// L := LEN(str);
// FOR pos := 1 TO L DO
// 	IF NOT ISC_ALPHA(pt^) THEN
// 		IS_ALPHA := FALSE;
// 		RETURN;
// 	END_IF;
//     	PT := PT + 1;
// END_FOR;
// IS_ALPHA := L > 0;
// END_FUNCTION

FUNCTION IS_CC : BOOL
VAR_INPUT
	str : STRING(STRING_LENGTH);
	cmp : STRING(STRING_LENGTH);
END_VAR
VAR
	L: INT;
	pos: INT;
END_VAR

L := LEN(str);
FOR pos := 1 TO L DO
	IF FIND(CMP,MID(str,1,pos)) = 0 THEN RETURN; END_IF;
END_FOR;
IS_CC := L > 0;
END_FUNCTION

// Commented out for beedance: it reads or writes the bytes of a STRING through a pointer; a beedance reference (REF_TO) refers to a whole variable of its type.
// FUNCTION IS_CTRL : BOOL
// VAR_INPUT
// 	STR : STRING(STRING_LENGTH);
// END_VAR
// VAR
// 	L: INT;
// 	pt : REF_TO BYTE;
// 	pos: INT;
// END_VAR
//
// PT := REF(str);
// L := LEN(str);
// FOR pos := 1 TO L DO
// 	IF NOT (ISC_CTRL(pt^)) THEN
// 		IS_CTRL := FALSE;
// 		RETURN;
// 	END_IF;
//     	PT := PT + 1;
// END_FOR;
// IS_CTRL := L > 0;
// END_FUNCTION

// Commented out for beedance: it reads or writes the bytes of a STRING through a pointer; a beedance reference (REF_TO) refers to a whole variable of its type.
// FUNCTION IS_HEX : BOOL
// VAR_INPUT
// 	str : STRING(STRING_LENGTH);
// END_VAR
// VAR
// 	L: INT;
// 	pt : REF_TO BYTE;
// 	pos: INT;
// END_VAR
//
// PT := REF(str);
// L := LEN(str);
// FOR pos := 1 TO L DO
// 	IF NOT (ISC_HEX(pt^)) THEN
// 		IS_HEX := FALSE;
// 		RETURN;
// 	END_IF;
//     	PT := PT + 1;
// END_FOR;
// IS_HEX := L > 0;
// END_FUNCTION

// Commented out for beedance: it reads or writes the bytes of a STRING through a pointer; a beedance reference (REF_TO) refers to a whole variable of its type.
// FUNCTION IS_LOWER : BOOL
// VAR_INPUT
// 	str : STRING(STRING_LENGTH);
// END_VAR
// VAR
// 	l: INT;
// 	pt : REF_TO BYTE;
// 	pos: INT;
// END_VAR
//
// PT := REF(str);
// L := LEN(str);
// FOR pos := 1 TO L DO
// 	IF NOT (ISC_LOWER(pt^)) THEN
// 		IS_LOWER := FALSE;
// 		RETURN;
// 	END_IF;
//     	PT := PT + 1;
// END_FOR;
// IS_LOWER := L > 0;
// END_FUNCTION

FUNCTION IS_NCC : BOOL
VAR_INPUT
	str : STRING(STRING_LENGTH);
	cmp : STRING(STRING_LENGTH);
END_VAR
VAR
	L: INT;
	pos: INT;
END_VAR

L := LEN(str);
FOR pos := 1 TO L DO
	IF FIND(CMP,MID(str,1,pos)) > 0 THEN RETURN; END_IF;
END_FOR;
IS_NCC := TRUE;
END_FUNCTION

// Commented out for beedance: it reads or writes the bytes of a STRING through a pointer; a beedance reference (REF_TO) refers to a whole variable of its type.
// FUNCTION IS_NUM : BOOL
// VAR_INPUT
// 	str : STRING(STRING_LENGTH);
// END_VAR
// VAR
// 	L : INT;
// 	pt : REF_TO BYTE;
// 	pos: INT;
// END_VAR
//
// PT := REF(str);
// L := LEN(str);
// FOR pos := 1 TO L DO
// 	IF NOT (ISC_NUM(pt^)) THEN
// 		IS_NUM := FALSE;
// 		RETURN;
// 	END_IF;
//     	PT := PT + 1;
// END_FOR;
// IS_NUM := L > 0;
// END_FUNCTION

// Commented out for beedance: it reads or writes the bytes of a STRING through a pointer; a beedance reference (REF_TO) refers to a whole variable of its type.
// FUNCTION IS_UPPER : BOOL
// VAR_INPUT
// 	str : STRING(STRING_LENGTH);
// END_VAR
// VAR
// 	L: INT;
// 	pt : REF_TO BYTE;
// 	pos: INT;
// END_VAR
//
// PT := REF(str);
// L := LEN(str);
// FOR pos := 1 TO L DO
// 	IF NOT (ISC_UPPER(pt^)) THEN
// 		IS_UPPER := FALSE;
// 		RETURN;
// 	END_IF;
//     	PT := PT + 1;
// END_FOR;
// IS_UPPER := L > 0;
// END_FUNCTION

FUNCTION ISC_ALPHA : BOOL
VAR_INPUT
	IN : BYTE;
END_VAR

IF setup.EXTENDED_ASCII THEN
	ISC_ALPHA := (in > 64 AND in < 91) OR (in > 191  AND in <> 215 AND in <> 247) OR (in > 96 AND in < 123);
ELSE
	ISC_ALPHA := (IN > 64 AND IN < 91) OR (in > 96 AND in < 123);
END_IF;
END_FUNCTION

FUNCTION ISC_CTRL : BOOL
VAR_INPUT
	IN : BYTE;
END_VAR

ISC_CTRL := IN < 32 OR IN = 127;
END_FUNCTION

FUNCTION ISC_HEX : BOOL
VAR_INPUT
	IN : BYTE;
END_VAR

ISC_HEX := (IN > 47 AND IN < 58) OR (IN > 64 AND IN < 71) OR (IN > 96 AND IN < 103);
END_FUNCTION

FUNCTION ISC_LOWER : BOOL
VAR_INPUT
	IN : BYTE;
END_VAR

IF setup.EXTENDED_ASCII THEN
	ISC_LOWER := ((in > 96) AND (in < 123)) OR ((in > 222) AND (in <> 247));
ELSE
	ISC_LOWER := ((in > 96) AND (in < 123));
END_IF;
END_FUNCTION

FUNCTION ISC_NUM : BOOL
VAR_INPUT
	IN : BYTE;
END_VAR

ISC_NUM := IN > 47 AND IN < 58;
END_FUNCTION

FUNCTION ISC_UPPER : BOOL
VAR_INPUT
	IN : BYTE;
END_VAR

IF setup.EXTENDED_ASCII THEN
	ISC_UPPER :=  ((in > 64) AND (in < 91)) OR (((in > 191) AND (in < 223)) AND (in <> 215));
ELSE
	ISC_UPPER := ((in > 64) AND (in < 91));
END_IF;
END_FUNCTION

// Commented out for beedance: it computes with pointers as addresses (pt := pt + 1); beedance references (REF_TO) have no arithmetic.
// FUNCTION LOWERCASE : STRING(STRING_LENGTH)
// VAR_INPUT
// 	str : STRING(STRING_LENGTH);
// END_VAR
// VAR
// 	PT : REF_TO BYTE;
// 	pos: INT;
// 	l: INT;
// END_VAR
//
// PT := REF(LOWERCASE);
// lowercase := str;
// l := LEN(str);
// FOR pos := 1 TO l DO
// 	pt^ := TO_LOWER(pt^);
// 	PT := PT + 1;
// END_FOR;
// END_FUNCTION

FUNCTION_BLOCK MESSAGE_4R
VAR_INPUT
	M0 : STRING(STRING_LENGTH);
	M1 : STRING(STRING_LENGTH);
	M2 : STRING(STRING_LENGTH);
	M3 : STRING(STRING_LENGTH);
	MM : INT := 3;
	ENQ : BOOL := TRUE;
	CLK : BOOL := TRUE;
	T1 : TIME := T#3s;
END_VAR
VAR_OUTPUT
	MX : STRING(STRING_LENGTH);
	MN : INT;
	TR : BOOL;
END_VAR
VAR
	timer : TON;
	edge: BOOL;
END_VAR

(* check for rising edge on EN *)
TR := FALSE;
IF ENQ THEN
	IF (NOT edge AND clk) OR timer.q THEN
			MN := INC1(MN, MM);
			TR := TRUE;
			timer(in := FALSE);
			CASE MN OF
				0 : MX := M0;
				1 : MX := M1;
				2 : MX := M2;
				3 : MX := M3;
			END_CASE;
	END_IF;
	edge := clk;
	timer( in := CLK, pt := T1);
ELSE
	MX := '';
	MN := 0;
END_IF;
END_FUNCTION_BLOCK

FUNCTION_BLOCK MESSAGE_8
VAR_INPUT
	IN1 : BOOL;
	IN2 : BOOL;
	IN3 : BOOL;
	IN4 : BOOL;
	IN5 : BOOL;
	IN6 : BOOL;
	IN7 : BOOL;
	IN8 : BOOL;
END_VAR
VAR_INPUT CONSTANT
	S1 : STRING(STRING_LENGTH);
	S2 : STRING(STRING_LENGTH);
	S3 : STRING(STRING_LENGTH);
	S4 : STRING(STRING_LENGTH);
	S5 : STRING(STRING_LENGTH);
	S6 : STRING(STRING_LENGTH);
	S7 : STRING(STRING_LENGTH);
	S8 : STRING(STRING_LENGTH);
END_VAR
VAR_OUTPUT
	M : STRING(STRING_LENGTH);
END_VAR

(* check if an alarm is present if yes set the output M otherwise clear M *)
IF in1 THEN
	M := S1;
ELSIF in2 THEN
	M := S2;
ELSIF in3 THEN
	M := S3;
ELSIF in4 THEN
	M := S4;
ELSIF in5 THEN
	M := S5;
ELSIF in6 THEN
	M := S6;
ELSIF in7 THEN
	M := S7;
ELSIF in8 THEN
	M := S8;
ELSE
	M := '';
END_IF;
END_FUNCTION_BLOCK

// Commented out for beedance: it reads or writes the bytes of a STRING through a pointer; a beedance reference (REF_TO) refers to a whole variable of its type.
// FUNCTION MIRROR : STRING(STRING_LENGTH)
// VAR_INPUT
// 	str : STRING(STRING_LENGTH);
// END_VAR
// VAR
// 	pi : REF_TO ARRAY[1..255] OF BYTE;
// 	po : REF_TO BYTE;
// 	lx: INT;
// 	i: INT;
// END_VAR
//
// pi := REF(str);
// po := REF(mirror);
// lx := LEN(str);
// FOR i := lx TO 1 BY - 1 DO
// 	po^ := pi^[i];
// 	po := po + 1;
// END_FOR;
// (* close output string *)
// po^:= 0;
// END_FUNCTION

FUNCTION MONTH_TO_STRING : STRING(10)
VAR_INPUT
	MTH : INT;
	LANG : INT;
	LX : INT;
END_VAR
VAR
	ly : INT;
END_VAR

IF LANG <= 0 THEN Ly := LANGUAGE.DEFAULT; ELSE ly := MIN(LANG, language.LMAX); END_IF;
IF MTH < 1 OR MTH > 12 THEN
	RETURN;
ELSIF LX = 0 THEN
	MONTH_TO_STRING := language.MONTHS[ly, MTH];
ELSIF Lx = 3 THEN
	MONTH_TO_STRING := language.MONTHS3[ly, MTH];
END_IF;
END_FUNCTION

// Commented out for beedance: it reads or writes the bytes of a STRING through a pointer; a beedance reference (REF_TO) refers to a whole variable of its type.
// FUNCTION OCT_TO_BYTE : BYTE
// VAR_INPUT
// 	OCT : STRING(10);
// END_VAR
// VAR
// 	pt : REF_TO BYTE;
// 	i: INT;
// 	X: BYTE;
// 	stop: INT;
// END_VAR
//
// pt := REF(oct);
// stop := LEN(oct);
// FOR I := 1 TO stop DO
// 	(* read the first character and subtract 48 to get value in decimal 0 = 48 *)
// 	x := pt^;
// 	(* calculate the value of the digit *)
// 	IF X > 47 AND x < 56 THEN
// 		OCT_TO_BYTE := SHL(OCT_TO_BYTE,3) + X - 48;
// 	END_IF;
// 	pt := pt + 1;
// END_FOR;
// END_FUNCTION

// Commented out for beedance: it reads or writes the bytes of a STRING through a pointer; a beedance reference (REF_TO) refers to a whole variable of its type.
// FUNCTION OCT_TO_DWORD : DWORD
// VAR_INPUT
// 	OCT : STRING(20);
// END_VAR
// VAR
// 	pt : REF_TO BYTE;
// 	i: INT;
// 	X: BYTE;
// 	stop: INT;
// END_VAR
//
// pt := REF(oct);
// stop := LEN(oct);
// FOR I := 1 TO stop DO
// 	(* read the first character and subtract 48 to get value in decimal 0 = 48 *)
// 	x := pt^;
// 	(* calculate the value of the digit *)
// 	IF X > 47 AND x < 56 THEN
// 		OCT_TO_DWORD := SHL(OCT_TO_DWORD,3) + X - 48;
// 	END_IF;
// 	pt := pt + 1;
// END_FOR;
// END_FUNCTION

FUNCTION REAL_TO_STRF : STRING(20)
VAR_INPUT
	IN : REAL;
	N : INT;
	D : STRING(1);
END_VAR
VAR
	O: REAL;
	i: INT;
END_VAR
VAR
	N_work : INT;
END_VAR
(* IEC 61131-3 does not let a POU assign to its inputs, so the body works on copies. *)
N_work := N;

(* LIMIT N to 0 .. 7 *)
N_work := LIMIT(0,N_work,7);
(* round the input to N digits and convert to string *)
O := ABS(in) * EXP10(N_work);
REAL_TO_STRF := DINT_TO_STRING(REAL_TO_DINT(O));
(* add zeroes in front to make sure sting is at least 8 digits long *)
FOR i := LEN(REAL_TO_STRF) TO N_work DO REAL_TO_STRF := CONCAT('0', REAL_TO_STRF); END_FOR;
(* add a dot if n > 0 *)
IF N_work > 0 THEN REAL_TO_STRF := INSERT(REAL_TO_STRF, D, LEN(REAL_TO_STRF) - N_work); END_IF;
(* add a minus sign if in is negative *)
IF in < 0 THEN REAL_TO_STRF := CONCAT('-', REAL_TO_STRF); END_IF;
END_FUNCTION

FUNCTION REPLACE_ALL : STRING(STRING_LENGTH)
VAR_INPUT
	str : STRING(STRING_LENGTH);
	src : STRING(STRING_LENGTH);
	rep : STRING(STRING_LENGTH);
END_VAR
VAR
	pos: INT;
	lp : INT;
	lx : INT;
END_VAR

REPLACE_ALL := str;
lx := LEN(src);
lp := LEN(rep);
pos := FINDP(REPLACE_ALL, src, 1);
WHILE pos > 0 DO
	REPLACE_ALL := REPLACE(REPLACE_ALL,rep,lx, pos);
	pos := FINDP(REPLACE_ALL, src, pos + lp);
END_WHILE;
END_FUNCTION

FUNCTION REPLACE_CHARS : STRING(STRING_LENGTH)
VAR_INPUT
	STR : STRING(STRING_LENGTH);
	SRC : STRING;
	REP : STRING;
END_VAR
VAR
	a, b : INT;
	c: STRING(1);
	stp: INT;
END_VAR
VAR
	SRC_work : STRING;
	REP_work : STRING;
END_VAR
(* IEC 61131-3 does not let a POU assign to its inputs, so the body works on copies. *)
SRC_work := SRC;
REP_work := REP;

REPLACE_CHARS := STR;
(* make sure rep and src are of same length and length is > 0 *)
a := LEN(SRC_work);
b := LEN(REP_work);
IF a < b THEN
	REP_work := LEFT(REP_work, a);
ELSIF b < a THEN
	SRC_work := LEFT(SRC_work, b);
END_IF;

(* search the string and replace if necessary *)
stp := LEN(str);
FOR a := 1 TO stp DO
	c := MID(REPLACE_CHARS, 1, a);
	b := FIND(SRC_work, c);
	IF b > 0 THEN
		REPLACE_CHARS := REPLACE(REPLACE_CHARS, MID(REP_work, 1, b), 1, a);
	END_IF;
END_FOR;
END_FUNCTION

// Commented out for beedance: it reads or writes the bytes of a STRING through a pointer; a beedance reference (REF_TO) refers to a whole variable of its type.
// FUNCTION REPLACE_UML : STRING(STRING_LENGTH)
// VAR_INPUT
// 	str : STRING(STRING_LENGTH);
// END_VAR
// VAR
// 	L : INT;
// 	pt : REF_TO BYTE;
// 	pto : REF_TO BYTE;
// 	ptm : REF_TO BYTE;
// 	pt1, pt2 : REF_TO BYTE;
// 	su : STRING(2);
// 	pos : INT;
// END_VAR
//
// PT := REF(str);
// pto := REF(REPLACE_UML);
// ptm := pto + INT_TO_DWORD(string_length);
// pt1 := REF(su);
// pt2 := pt1 + 1;
// L := LEN(str);
// WHILE pos < L AND pos < string_length DO
// 	IF pt^ < 127 THEN
// 		(* no uml character simlply copy the character*)
// 		pto^ := pt^;
// 	ELSE
// 		(* convert the uml character *)
// 		su := TO_UML(pt^);
// 		(* we must make sure pointer are not out of range *)
// 		pto^ := pt1^;
// 		IF pto < ptm AND pt2^ > 0 THEN
// 			pto := pto + 1;
// 			pto^ := pt2^;
// 		END_IF;
// 	END_IF;
// 	(* increment pointers *)
// 	pt := pt + 1;
// 	pto := pto + 1;
// 	pos := pos + 1;
// END_WHILE;
//
// (* properly close the output string *)
// pto^ := 0;
// END_FUNCTION

FUNCTION_BLOCK TICKER

VAR_INPUT
	N : INT;
	PT : TIME;
END_VAR

VAR_IN_OUT
	Text : STRING(STRING_LENGTH);
END_VAR

VAR_OUTPUT
	Display : STRING(STRING_LENGTH);
END_VAR
VAR
	delay : TP;
	step : INT;
END_VAR

(* generate next ticker when delay is low *)
IF N < LEN(text) THEN
	IF NOT delay.Q THEN
		(* increase step for next tick *)
		step := step + 1;
		IF step > LEN(text) THEN step := 1; END_IF;
		(* extract dispay from text *)
		display := MID(text, N, step);
		(* set delay timer for next tick *)
		delay(in := TRUE, PT := PT);
	ELSE;
		(* execute delay timer *)
		delay(in := FALSE);
	END_IF;
ELSE
	display := text;
END_IF;
END_FUNCTION_BLOCK

FUNCTION TO_LOWER : BYTE
VAR_INPUT
	IN : BYTE;
END_VAR

IF in > 64 AND in < 91 THEN
   TO_LOWER := in OR 16#20;
ELSIF (in > 191 AND in < 223) AND in <> 215 AND setup.EXTENDED_ASCII THEN
   TO_LOWER := in OR 16#20;
ELSE
   TO_LOWER := in;
END_IF;
END_FUNCTION

// Commented out for beedance: it uses CHR_TO_STRING, which is commented out.
// FUNCTION TO_UML : STRING(2)
// VAR_INPUT
// 	IN : BYTE;
// END_VAR
//
// CASE in OF
// 	196:	(* Ä *)
// 		TO_UML := 'Ae';
// 	214:	(* Ö *)
// 		TO_UML := 'Oe';
// 	220:	(* Ü *)
// 		TO_UML := 'Ue';
// 	223:	(* ß *)
// 		TO_UML := 'ss';
// 	228:	(* ä *)
// 		TO_UML := 'ae';
// 	246:	(* ö *)
// 		TO_UML := 'oe';
// 	252:	(* ü *)
// 		TO_UML := 'ue';
// ELSE
// 	TO_UML := CHR_TO_STRING(IN);
// END_CASE;
// END_FUNCTION

FUNCTION TO_UPPER : BYTE
VAR_INPUT
	IN : BYTE;
END_VAR

IF in > 96 AND in < 123 THEN
   TO_UPPER := in AND 16#DF;
ELSIF in > 223 AND in <> 247 AND in <> 255 AND setup.EXTENDED_ASCII THEN
   TO_UPPER := in AND 16#DF;
ELSE
   TO_UPPER := in;
END_IF;
END_FUNCTION

FUNCTION TRIM : STRING(STRING_LENGTH)
VAR_INPUT
	str : STRING(STRING_LENGTH);
END_VAR
VAR
	pos: INT;
END_VAR

TRIM := str;
REPEAT
	pos := FIND(trim,' ');
	IF pos > 0 THEN TRIM := REPLACE(TRIM,'',1,pos); END_IF;
UNTIL pos = 0	END_REPEAT;
END_FUNCTION

FUNCTION TRIM1 : STRING(STRING_LENGTH)
VAR_INPUT
	str : STRING(STRING_LENGTH);
END_VAR
VAR
	pos: INT;
END_VAR

TRIM1 := str;
REPEAT
	pos := FIND(trim1,'  ');
	IF pos > 0 THEN TRIM1 := REPLACE(TRIM1,' ',2,pos); END_IF;
UNTIL pos = 0	END_REPEAT;
(* beginning and ending blanks need to be stripped off *)
IF LEFT(trim1,1) = ' ' THEN trim1 := DELETE(trim1,1,1); END_IF;
IF RIGHT(trim1,1) = ' ' THEN trim1 := DELETE(trim1,1,LEN(trim1)); END_IF;
END_FUNCTION

FUNCTION TRIME : STRING(string_length)
VAR_INPUT
	str : STRING(STRING_LENGTH);
END_VAR

TRIME := str;
(* beginning blanks need to be stripped off *)
WHILE LEFT(TRIME,1) = ' ' DO
	TRIME := DELETE(TRIME,1,1);
END_WHILE;

(* ending blanks need to be stripped off *)
WHILE RIGHT(TRIME,1) = ' ' DO
	TRIME := DELETE(TRIME,1,LEN(TRIME));
END_WHILE;
END_FUNCTION

// Commented out for beedance: it computes with pointers as addresses (pt := pt + 1); beedance references (REF_TO) have no arithmetic.
// FUNCTION UPPERCASE : STRING(STRING_LENGTH)
// VAR_INPUT
// 	str : STRING(STRING_LENGTH);
// END_VAR
// VAR
// 	pt : REF_TO BYTE;
// 	pos: INT;
// 	l: INT;
// END_VAR
//
// pt := REF(UPPERCASE);
// UPPERCASE := str;
// l := LEN(str);
// FOR pos := 1 TO l DO
// 	pt^ := TO_UPPER(pt^);
// 	pt := pt + 1;
// END_FOR;
// END_FUNCTION

FUNCTION WEEKDAY_TO_STRING : STRING(10)
VAR_INPUT
	WDAY : INT;
	LANG : INT;
	LX : INT;
END_VAR
VAR
	ly : INT;
END_VAR

IF LANG <= 0 THEN ly := LANGUAGE.DEFAULT; ELSE ly := MIN(LANG, LANGUAGE.LMAX); END_IF; (* OSCAT 3.36 *)
IF wday < 1 OR wday > 7 THEN
	RETURN;
ELSIF LX = 0 THEN
	WEEKDAY_TO_STRING := language.WEEKDAYS[ly, WDAY];
ELSIF Lx = 2 THEN
	WEEKDAY_TO_STRING := language.WEEKDAYS2[ly, WDAY];
END_IF;
END_FUNCTION

FUNCTION_BLOCK CALENDAR_CALC
VAR_INPUT
	SPE : BOOL;
	H : REAL := -0.83333333333;
END_VAR
VAR_IN_OUT
	XCAL : CALENDAR;
	HOLIDAYS : ARRAY[0..29] OF HOLIDAY_DATA;
END_VAR
VAR
	last : DT;
	last_day : DINT;
	holy : HOLIDAY;
	sun : SUN_TIME;
	last_hour: INT;
	utod: TOD;
	pos : SUN_POS;
	plast: DT;
END_VAR
VAR_TEMP
	dtemp : DINT;
	tmp : INT;
END_VAR

IF xcal.UTC <> last THEN
	(* run once per second *)
	(* update utc last calculated  *)
	last := XCAL.UTC;
	utod := DT_TO_TOD(xcal.UTC);

	(* calculate ltc from utc *)
	XCAL.LOCAL_DT := UTC_TO_LTIME(XCAL.UTC, XCAL.DST_EN, XCAL.OFFSET);
	XCAL.LOCAL_DATE := DT_TO_DATE(XCAL.LOCAL_DT);
	XCAL.LOCAL_TOD := DT_TO_TOD(XCAL.LOCAL_DT);
	dtemp := DAY_OF_DATE(XCAL.LOCAL_DATE);
	xcal.night := XCAL.LOCAL_TOD < XCAL.SUN_RISE OR XCAL.LOCAL_TOD > XCAL.SUN_SET;

	(* run once per hour *)
	tmp := HOUR(xcal.LOCAL_TOD);
	IF  tmp <> last_hour THEN
		XCAL.DST_ON := DST(XCAL.UTC) AND xcal.DST_EN;
		last_hour := tmp;
	END_IF;

	(* run once per day *)
	IF dtemp <> last_day THEN
		last_day := dtemp;
		(* a new day has started, recalculate daily events *)
		XCAL.YEAR := YEAR_OF_DATE(XCAL.LOCAL_DATE);
		XCAL.MONTH := MONTH_OF_DATE(XCAL.LOCAL_DATE);
		XCAL.DAY := DAY_OF_MONTH(XCAL.LOCAL_DATE);
		XCAL.WEEKDAY := DAY_OF_WEEK(XCAL.LOCAL_DATE);
		HOLY(date_in := XCAL.LOCAL_DATE, LANGU := xcal.LANGUAGE, HOLIDAYS := HOLIDAYS);
		XCAL.HOLIDAY := HOLY.Y;
		XCAL.HOLY_NAME := HOLY.NAME;
		sun(latitude := XCAL.LATITUDE, longitude := xcal.LONGITUDE, utc := DT_TO_DATE(xcal.UTC), H := H);
		XCAL.SUN_RISE := DINT_TO_TOD(TOD_TO_DINT(sun.sun_rise) + XCAL.OFFSET * 60000 + SEL(XCAL.DST_ON,DINT#0,3600000));
		XCAL.SUN_SET := DINT_TO_TOD(TOD_TO_DINT(sun.sun_set) + XCAL.OFFSET * 60000 + SEL(XCAL.DST_ON,DINT#0,3600000));
		XCAL.SUN_MIDDAY := DINT_TO_TOD(TOD_TO_DINT(sun.MIDDAY) + XCAL.OFFSET * 60000 + SEL(XCAL.DST_ON,DINT#0,3600000));
		XCAL.SUN_HEIGTH := sun.sun_declination;
		XCAL.WORK_WEEK := WORK_WEEK(XCAL.LOCAL_DATE);
	END_IF;

	(* calculate the suns position every 10 seconds when SPE = TRUE *)
	IF SPE AND xcal.UTC -  plast >= t#25s THEN
		plast := last;
		pos(latitude := xcal.LATITUDE, longitude := xcal.LONGITUDE, utc := xcal.UTC);
		xcal.SUN_HOR := pos.B;
		xcal.SUN_VER := pos.HR;
	END_IF;
END_IF;
END_FUNCTION_BLOCK

FUNCTION DATE_ADD : DATE
VAR_INPUT
	IDATE : DATE;
	D : INT;
	W : INT;
	M : INT;
	Y : INT;
END_VAR
VAR
	mo: INT;
	yr : INT;
	dm: INT;
END_VAR

DATE_ADD := UDINT_TO_DATE(DATE_TO_UDINT(IDATE) + INT_TO_UDINT(D + W * 7) * UDINT#86400);
yr := Y + YEAR_OF_DATE(DATE_ADD);
mo := M + MONTH_OF_DATE(DATE_ADD);
dm := DAY_OF_MONTH(DATE_ADD);
WHILE mo > 12 DO
	mo := mo - 12;
	yr := yr + 1;
END_WHILE;
WHILE mo < 1 DO
	mo := mo + 12;
	yr := yr - 1;
END_WHILE;
DATE_ADD := SET_DATE(yr, mo, dm);
END_FUNCTION

FUNCTION DAY_OF_DATE : DINT
VAR_INPUT
	idate : DATE;
END_VAR

DAY_OF_DATE := UDINT_TO_DINT(DATE_TO_UDINT(idate) / 86400);
END_FUNCTION

FUNCTION DAY_OF_MONTH : INT
VAR_INPUT
	IDATE : DATE;
END_VAR
VAR
	leap: INT;
END_VAR

(* calculate the day in the year *)
DAY_OF_MONTH := DAY_OF_YEAR(idate);
(* leap will be set to one for a leap year *)
leap := BOOL_TO_INT(LEAP_OF_DATE(idate));
(* if leap year deduct one from the days of the year *)
DAY_OF_MONTH := DAY_OF_MONTH - leap;
(* search if we are in month december to march ? *)
IF DAY_OF_MONTH > setup.MTH_OFS[9] THEN
	IF DAY_OF_MONTH > setup.MTH_OFS[11] THEN
		IF DAY_OF_MONTH > setup.mth_ofs[12] THEN
			DAY_OF_MONTH := DAY_OF_MONTH - setup.MTH_OFS[12];
		ELSE
			DAY_OF_MONTH := DAY_OF_MONTH - setup.MTH_OFS[11];
		END_IF;
	ELSE
		IF DAY_OF_MONTH > setup.mth_ofs[10] THEN
			DAY_OF_MONTH := DAY_OF_MONTH - setup.MTH_OFS[10];
		ELSE
			DAY_OF_MONTH := DAY_OF_MONTH - setup.MTH_OFS[9];
		END_IF;
	END_IF;
ELSIF DAY_OF_MONTH > setup.MTH_OFS[5] THEN
	IF DAY_OF_MONTH > setup.MTH_OFS[7] THEN
		IF DAY_OF_MONTH > setup.mth_ofs[8] THEN
			DAY_OF_MONTH := DAY_OF_MONTH - setup.MTH_OFS[8];
		ELSE
			DAY_OF_MONTH := DAY_OF_MONTH - setup.MTH_OFS[7];
		END_IF;
	ELSE
		IF DAY_OF_MONTH > setup.mth_ofs[6] THEN
			DAY_OF_MONTH := DAY_OF_MONTH - setup.MTH_OFS[6];
		ELSE
			DAY_OF_MONTH := DAY_OF_MONTH - setup.MTH_OFS[5];
		END_IF;
	END_IF;
ELSIF DAY_OF_MONTH > setup.MTH_OFS[3] THEN
	IF DAY_OF_MONTH > setup.MTH_OFS[4] THEN
		DAY_OF_MONTH := DAY_OF_MONTH - setup.MTH_OFS[4];
	ELSE
		DAY_OF_MONTH := DAY_OF_MONTH - setup.MTH_OFS[3];
	END_IF;
ELSE
	(* since now we must be in february or january we need to add leap again *)
	DAY_OF_MONTH := DAY_OF_MONTH + leap;
	IF DAY_OF_MONTH > setup.MTH_OFS[2] THEN DAY_OF_MONTH := DAY_OF_MONTH - setup.mth_ofs[2]; END_IF;
	(* since nothing was true before, day_of_month must already be good *)
END_IF;
END_FUNCTION

FUNCTION DAY_OF_WEEK : INT
VAR_INPUT
	IDATE : DATE;
END_VAR

DAY_OF_WEEK := UDINT_TO_INT((DATE_TO_UDINT(idate) / 86400 + 3) MOD 7) + 1;
END_FUNCTION

FUNCTION DAY_OF_YEAR : INT
VAR_INPUT
	IDATE : DATE;
END_VAR

DAY_OF_YEAR := UDINT_TO_INT((DATE_TO_UDINT(idate) / UDINT#86400) MOD UDINT#1461);
IF DAY_OF_YEAR > 729 THEN
	IF DAY_OF_YEAR > 1095 THEN DAY_OF_YEAR := DAY_OF_YEAR - 1095; ELSE DAY_OF_YEAR := DAY_OF_YEAR - 729; END_IF;
ELSIF DAY_OF_YEAR > 364 THEN
	DAY_OF_YEAR := DAY_OF_YEAR - 364;
ELSE
	DAY_OF_YEAR := DAY_OF_YEAR + 1;
END_IF;
END_FUNCTION

FUNCTION DAY_TO_TIME : TIME
VAR_INPUT
	IN : REAL;
END_VAR

DAY_TO_TIME := DWORD_TO_TIME(REAL_TO_DWORD(IN * 86400000.0));
END_FUNCTION

FUNCTION DAYS_DELTA : DINT
VAR_INPUT
	date_1 : DATE;
	date_2 : DATE;
END_VAR

IF DATE_1 > DATE_2 THEN
	DAYS_DELTA := - UDINT_TO_DINT((DATE_TO_UDINT(date_1) - DATE_TO_UDINT(date_2)) / 86400);
ELSE
	DAYS_DELTA := UDINT_TO_DINT((DATE_TO_UDINT(date_2) - DATE_TO_UDINT(date_1)) / 86400);
END_IF;
END_FUNCTION

FUNCTION DAYS_IN_MONTH : INT
VAR_INPUT
	IDATE : DATE;
END_VAR

DAYS_IN_MONTH := DAY_OF_YEAR(IDATE);
IF LEAP_OF_DATE(IDATE) THEN
	CASE DAYS_IN_MONTH OF
		32..60	:	DAYS_IN_MONTH := 29;
		92..121 :	DAYS_IN_MONTH := 30;
		153..182:	DAYS_IN_MONTH := 30;
		245..274:	DAYS_IN_MONTH := 30;
		306..335:	DAYS_IN_MONTH := 30;
	ELSE
		DAYS_IN_MONTH := 31;
	END_CASE;
ELSE
	CASE DAYS_IN_MONTH OF
		32..59	:	DAYS_IN_MONTH := 28;
		91..120 :	DAYS_IN_MONTH := 30;
		152..181:	DAYS_IN_MONTH := 30;
		244..273:	DAYS_IN_MONTH := 30;
		305..334:	DAYS_IN_MONTH := 30;
	ELSE
		DAYS_IN_MONTH := 31;
	END_CASE;
END_IF;
END_FUNCTION

FUNCTION DAYS_IN_YEAR : INT
VAR_INPUT
	IDATE : DATE;
END_VAR

IF LEAP_OF_DATE(IDATE) THEN
	DAYS_IN_YEAR := 366;
ELSE
	DAYS_IN_YEAR := 365;
END_IF;
END_FUNCTION

FUNCTION_BLOCK DCF77
VAR_INPUT
	REC : BOOL;
	SET : BOOL;
	SDT : DT;
	DSI : BOOL;
END_VAR
VAR_INPUT CONSTANT
	SYNC_TIMEOUT : TIME := t#2m;
	TIME_OFFSET : INT := 1;
	DST_EN : BOOL := TRUE;
END_VAR
VAR_OUTPUT
	TP : BOOL;
	DS : BOOL;
	WDAY : INT;
	ERROR : BOOL := TRUE;
	RTC : DT;
	RTC1 : DT;
	MSEC : INT;
	SYNC : BOOL;
END_VAR
VAR
	mez : DT;
	utc : DT;
	state : INT;
	edge: BOOL;
	tx : TIME;
	ty: TIME;
	last : TIME;
	bits : ARRAY[0..58] OF BOOL;
	cnt : INT;
	i : INT;
	old_time : DT;
	minute : INT;
	hour : INT;
	day : INT;
	month : INT;
	year : INT;
	last_sync: TIME;
	t1: TIME;
	tz: TIME;
	init: BOOL;
END_VAR

(* if tp was set it should only be active for 1 cycle *)
TP := FALSE;

(* read system time *)
t1 := DWORD_TO_TIME(T_PLC_MS());
tx := t1 - last;

IF rec XOR edge THEN
	edge := rec;
	IF NOT rec AND tx > t#1700ms AND tx < t#2000ms THEN
		(* start condition reached *)
		state := 0;
		tp := NOT error;
	ELSIF NOT rec AND tx > t#700ms AND tx < t#1000ms THEN
		(* second switch detected *)
		IF state < 58 THEN state := state +1; ELSE state := 0; END_IF;
	ELSIF rec AND tx  < t#120ms THEN
		(* bit 0 detected  *)
		bits[state] := 0;
	ELSIF rec AND tx > t#120ms AND tx < t#250ms THEN
		(* bit 1 detected *)
		bits[state] := 1;
	ELSE
		(* error condition received signal is not valid *)
		error := TRUE;
		state := 0;
	END_IF;
	last := last + tx;
	IF rec AND state = 58 THEN
		error := FALSE;

		(* decode the bits and check for possible errors *)
		IF bits[0] OR NOT (bits[17] XOR bits[18]) OR NOT bits[20] THEN error := TRUE; END_IF;
		(* decode minute *)
		MINUTE := 0;
		MINUTE.0 := bits[21];
		MINUTE.1 := bits[22];
		MINUTE.2 := bits[23];
		MINUTE.3 := bits[24];
		IF bits[25] THEN MINUTE := MINUTE + 10; END_IF;
		IF bits[26] THEN MINUTE := MINUTE + 20; END_IF;
		IF bits[27] THEN MINUTE := MINUTE + 40; END_IF;
		IF MINUTE > 59 OR (bits[21] XOR bits[22] XOR bits[23] XOR bits[24] XOR bits[25] XOR bits[26] XOR bits[27] XOR bits[28]) THEN error := TRUE; END_IF;

		(* decode hour *)
		HOUR := 0;
		HOUR.0 := bits[29];
		HOUR.1 := bits[30];
		HOUR.2 := bits[31];
		HOUR.3 := bits[32];
		IF bits[33] THEN HOUR := HOUR + 10; END_IF;
		IF bits[34] THEN HOUR := HOUR +20; END_IF;
		IF HOUR > 23 OR (bits[29] XOR bits[30] XOR bits[31] XOR bits[32] XOR bits[33] XOR bits[34] XOR bits[35]) THEN error := TRUE; END_IF;

		(* decode day of month *)
		day := 0;
		day.0 := bits[36];
		day.1 := bits[37];
		day.2 := bits[38];
		day.3 := bits[39];
		IF bits[40] THEN day := day + 10; END_IF;
		IF bits[41] THEN day := day + 20; END_IF;
		IF day > 31 THEN error := TRUE; END_IF;

		(* decode day of week *)
		wday := 0;
		wday.0 := bits[42];
		wday.1 := bits[43];
		wday.2 := bits[44];
		IF wday > 7 OR wday < 1 THEN error := TRUE; END_IF;

		(* decode month *)
		MONTH := 0;
		MONTH.0 := bits[45];
		MONTH.1 := bits[46];
		MONTH.2 := bits[47];
		MONTH.3 := bits[48];
		IF bits[49] THEN MONTH := MONTH +10; END_IF;
		IF MONTH > 12 THEN error := TRUE; END_IF;

		(* decode year *)
		YEAR := 0;
		YEAR.0 := bits[50];
		YEAR.1 := bits[51];
		YEAR.2 := bits[52];
		YEAR.3 := bits[53];
		IF bits[54] THEN YEAR := YEAR + 10; END_IF;
		IF bits[55] THEN YEAR := YEAR + 20; END_IF;
		IF bits[56] THEN YEAR := YEAR + 40; END_IF;
		IF bits[57] THEN YEAR := YEAR + 80; END_IF;

		(* check parity for bits 36 to 58 *)
		cnt := 0;
		FOR i := 36 TO 58 DO IF bits[i] THEN cnt := cnt + 1; END_IF; END_FOR;
		IF NOT EVEN(cnt) THEN error := TRUE; END_IF;

		(* time must be valid for two cycles to clear error flag *)
		IF NOT error THEN
			(* set outputs *)
			old_time := mez;
			IF YEAR >= 70 THEN YEAR := YEAR + 1900; ELSE YEAR := YEAR + 2000; END_IF;
			mez := SET_DT(YEAR,MONTH,day,HOUR,MINUTE,0);
			DS := bits[17];
			IF DS THEN
				UTC := UDINT_TO_DT(DT_TO_UDINT(mez) - 7200);
			ELSE
				UTC := UDINT_TO_DT(DT_TO_UDINT(mez) - 3600);
			END_IF;

			(* set trigger signal only if the receiver has received 2 successive minutes *)
			IF mez <> old_time + t#1m THEN error := TRUE ; END_IF;
		END_IF;
	END_IF;
END_IF;

(* this portion implements a free running clock which is triggered by the dcf77 signal *)
tz := UDINT_TO_TIME(INT_TO_UDINT(ABS(time_offset)) * 3600000);

(* input sdt is copied to utc at first power up *)
IF NOT init OR SET THEN
	init := TRUE;
	utc := sdt;
	tp := TRUE;
	DS := DSI;
END_IF;

IF tp THEN
	rtc := utc;
	IF DS AND dst_en THEN
		IF time_offset < 0 THEN	rtc1 := rtc - tz + t#1h; ELSE rtc1 := rtc + tz + t#1h; END_IF;
	ELSE
		IF time_offset < 0 THEN rtc1 := rtc - tz; ELSE rtc1 := rtc + tz; END_IF;
	END_IF;
	sync := TRUE;
	last_sync := last;
	ty := last;
ELSIF rtc > DWORD_TO_DT(0) AND T1 - ty >= t#1s THEN
	rtc := rtc + t#1s;
	rtc1 := rtc1 + t#1s;
	ty := ty + t#1s;
	sync := ty - last_sync < sync_timeout AND last_sync > DWORD_TO_TIME(0);
	wday := DAY_OF_WEEK(DT_TO_DATE(rtc1));
	DS := dst_en AND DST(utc);
END_IF;
msec := TIME_TO_INT(t1 - ty);
END_FUNCTION_BLOCK

FUNCTION DST : BOOL
VAR_INPUT
	UTC : DT;
END_VAR
VAR
	yr : INT;
	yr4 : DWORD;
	ltc: DWORD;
	idate : DWORD;
END_VAR

yr := YEAR_OF_DATE(DT_TO_DATE(UTC));
ltc := DT_TO_DWORD(UTC);
idate := DT_TO_DWORD(SET_DT(yr, 3, 31, 1, 0, 0));
yr4 := ULINT_TO_DWORD(INT_TO_ULINT(yr) * 5 / 4 + 1);
DST := (DWORD_TO_ULINT(idate) - ((DWORD_TO_ULINT(yr4) + 3) MOD 7) * 86400 <= DWORD_TO_ULINT(ltc)) AND (DWORD_TO_ULINT(idate) + (214 - DWORD_TO_ULINT(yr4) MOD 7) * 86400 > DWORD_TO_ULINT(ltc));
END_FUNCTION

FUNCTION DT2_TO_SDT : SDT
VAR_INPUT
	DI : DATE;
	TI : TOD;
END_VAR

DT2_TO_SDT.YEAR := YEAR_OF_DATE(di);
DT2_TO_SDT.MONTH := MONTH_OF_DATE(di);
DT2_TO_SDT.DAY := DAY_OF_MONTH(di);
DT2_TO_SDT.WEEKDAY := DAY_OF_WEEK(di);
DT2_TO_SDT.MS := UDINT_TO_INT(TOD_TO_UDINT(ti) MOD 1000);
DT2_TO_SDT.SECOND := UDINT_TO_INT((TOD_TO_UDINT(ti) / 1000) MOD 60);
DT2_TO_SDT.MINUTE := UDINT_TO_INT((TOD_TO_UDINT(ti) / 60000) MOD 60);
DT2_TO_SDT.HOUR := UDINT_TO_INT(TOD_TO_UDINT(ti) / 3600000);
END_FUNCTION

FUNCTION DT_TO_SDT : SDT
VAR_INPUT
	DTI : DT;
END_VAR
VAR
	tmp : DATE;
	tdt : DWORD;
END_VAR

tmp := DT_TO_DATE(dti);
tdt := ULINT_TO_DWORD(DT_TO_ULINT(dti) - DATE_TO_ULINT(tmp));
DT_TO_SDT.YEAR := YEAR_OF_DATE(tmp);
DT_TO_SDT.MONTH := MONTH_OF_DATE(tmp);
DT_TO_SDT.DAY := DAY_OF_MONTH(tmp);
DT_TO_SDT.WEEKDAY := DAY_OF_WEEK(tmp);
DT_TO_SDT.SECOND := ULINT_TO_INT(DWORD_TO_ULINT(tdt) MOD 60);
DT_TO_SDT.MINUTE := ULINT_TO_INT((DWORD_TO_ULINT(tdt) / 60) MOD 60);
DT_TO_SDT.HOUR := ULINT_TO_INT(DWORD_TO_ULINT(tdt) / 3600);
END_FUNCTION

FUNCTION EASTER : DATE
VAR_INPUT
	year : INT;
END_VAR
VAR
	b,c: INT;
	oday: INT;
END_VAR

b := (204 - 11 * (YEAR MOD 19)) MOD 30;
IF b > 27 THEN b := b - 1; END_IF;
c := (year + year / 4 + b - 13) MOD 7;
oday := 28 + b - c;
IF oday > 33 THEN
	EASTER := SET_DATE(year, 4, oday - 31);
ELSE
	EASTER := SET_DATE(year, 3, oday);
END_IF;
END_FUNCTION

FUNCTION_BLOCK EVENTS
VAR_INPUT
	DATE_IN : DATE;
	ENA : BOOL;
END_VAR
VAR_OUTPUT
	Y : BOOL;
	NAME : STRING(30);
END_VAR
VAR
	i : INT;
	last_active : DATE;
	size :INT := 49;
	day_in: DINT;
	cyr: INT;
	lday: DINT;
	check : HOLIDAY_DATA;
	y_int : BOOL;
	name_int : STRING(30);
END_VAR
VAR_IN_OUT
	ELIST : ARRAY[0..49] OF HOLIDAY_DATA;
END_VAR

(* for performance reasons only activate once a day *)
IF last_active <> date_in THEN
	last_active := DATE_IN;
	Y_int := FALSE;
	name_int := '';
	day_in := DAY_OF_DATE(DATE_IN);
	cyr := YEAR_OF_DATE(DATE_IN);

	(* search list for events *)
	FOR i := 0 TO size DO
		check := elist[i];
		lday := DAY_OF_DATE(SET_DATE(cyr,check.month, check.day));
		IF day_in >= lday AND day_in <= lday + check.use - 1 THEN
			y_int := TRUE;
			name_int := check.name;
			EXIT;
		END_IF;
	END_FOR;
END_IF;

IF ENA THEN
	Y := y_int;
	NAME := name_int;
ELSE
	Y := FALSE;
	NAME := '';
END_IF;
END_FUNCTION_BLOCK

FUNCTION_BLOCK HOLIDAY
VAR_INPUT
	DATE_IN : DATE;
	LANGU : INT;
	FRIDAY : BOOL;
	SATURDAY : BOOL;
	SUNDAY : BOOL;
END_VAR
VAR_IN_OUT
	HOLIDAYS : ARRAY[0..29] OF HOLIDAY_DATA;
END_VAR
VAR CONSTANT
	SIZE : INT := 29;
END_VAR
VAR_OUTPUT
	Y : BOOL;
	NAME : STRING(30);
END_VAR
VAR
	last_active : DATE;
	ostern: DATE;
	i: INT;
	jahr: INT;
	x_date: DATE;
	lx: INT;
	wdx: INT;
END_VAR

(* for performance reasons only activate once a day *)
IF last_active = date_in THEN RETURN; END_IF;
last_active := DATE_IN;

(* determine language *)
IF LANGU = 0 THEN
	lx := language.DEFAULT;
ELSE
	lx := MIN(language.LMAX, LANGU);
END_IF;

(* calculate easter for the current year *)
jahr := YEAR_OF_DATE(date_in);
ostern := EASTER(jahr);
wdx := DAY_OF_WEEK(DATE_IN);
Y := FALSE;

(* check for holidays *)
FOR i := 0 TO size DO
	x_date := SET_DATE(jahr, HOLIDAYS[i].MONTH , HOLIDAYS[i].DAY);
	IF HOLIDAYS[i].USE = 1 AND HOLIDAYS[i].MONTH > 0 THEN
		(* check for fixed date holiday *)
		IF x_date = date_in THEN
			Y := TRUE;
			NAME := HOLIDAYS[i].NAME;
			RETURN;
		END_IF;
	ELSIF HOLIDAYS[i].USE = 1 AND HOLIDAYS[i].MONTH = 0 THEN
		(* check for holiday in reference to easter *)
		IF DATE_ADD(ostern, HOLIDAYS[i].DAY ,0,0,0) = date_in THEN
			Y := TRUE;
			NAME := HOLIDAYS[i].NAME;
			RETURN;
		END_IF;
	ELSIF HOLIDAYS[i].USE < 0 THEN
		(* check for holiday on a weekday before date *)
		IF DAY_OF_WEEK(date_in) = ABS(HOLIDAYS[i].USE) AND date_in < x_date AND date_in >= DATE_ADD(x_date,-7,0,0,0) THEN
			Y := TRUE;
			NAME := HOLIDAYS[i].NAME;
			RETURN;
		END_IF;
	END_IF;
END_FOR;

(* check array if today is weekend *)
IF NOT Y AND (wdx = 5 AND FRIDAY OR wdx = 6 AND SATURDAY OR wdx = 7 AND SUNDAY) THEN
	Y := TRUE;
	NAME := LANGUAGE.WEEKDAYS[LOCATION.LANGUAGE[lx],wdx];
ELSE
	NAME := '';
END_IF;
END_FUNCTION_BLOCK

FUNCTION HOUR : INT
VAR_INPUT
	itod : TOD;
END_VAR

HOUR := UDINT_TO_INT(TOD_TO_UDINT(itod) / 3600000);
END_FUNCTION

FUNCTION HOUR_OF_DT : INT
VAR_INPUT
	XDT : DT;
END_VAR

HOUR_OF_DT := UDINT_TO_INT((DT_TO_UDINT(XDT) MOD 86400) / 3600);
END_FUNCTION

FUNCTION HOUR_TO_TIME : TIME
VAR_INPUT
	IN : REAL;
END_VAR

HOUR_TO_TIME := DWORD_TO_TIME(REAL_TO_DWORD(IN * 3600000));
END_FUNCTION

FUNCTION HOUR_TO_TOD : TOD
VAR_INPUT
	IN : REAL;
END_VAR

HOUR_TO_TOD := DWORD_TO_TOD(REAL_TO_DWORD(IN * 3600000));
END_FUNCTION

FUNCTION JD2000 : REAL
VAR_INPUT
	DTI : DT;
END_VAR

JD2000 := UDINT_TO_REAL(DT_TO_UDINT(DTI) - 946728000) / 86400.0;
END_FUNCTION

FUNCTION LEAP_DAY : BOOL
VAR_INPUT
	IDATE : DATE;
END_VAR
VAR
END_VAR

LEAP_DAY := DATE_TO_UDINT(IDATE) MOD 126230400 = 68169600;
END_FUNCTION

FUNCTION LEAP_OF_DATE : BOOL
VAR_INPUT
	idate : DATE;
END_VAR

LEAP_OF_DATE := SHL(UDINT_TO_DWORD((DATE_TO_UDINT(idate) + 43200) / 31557600), 30) = 16#80000000;
END_FUNCTION

FUNCTION LEAP_YEAR : BOOL
VAR_INPUT
	yr : INT;
END_VAR

LEAP_YEAR := yr MOD 4 = 0;
END_FUNCTION

FUNCTION LTIME_TO_UTC : DT
VAR_INPUT
	LTIME : DT;
	DST : BOOL;
	TIME_ZONE_OFFSET : INT;
END_VAR

LTIME_TO_UTC := UDINT_TO_DT(DT_TO_UDINT(LTIME) - INT_TO_UDINT(TIME_ZONE_OFFSET) * 60);
IF DST THEN LTIME_TO_UTC := LTIME_TO_UTC - T#1h; END_IF;
END_FUNCTION

FUNCTION MINUTE : INT
VAR_INPUT
	itod : TOD;
END_VAR

MINUTE := UDINT_TO_INT(TOD_TO_UDINT(itod) / 60000 - TOD_TO_UDINT(itod) / 3600000 * 60);
END_FUNCTION

FUNCTION MINUTE_OF_DT : INT
VAR_INPUT
	XDT : DT;
END_VAR

MINUTE_OF_DT := UDINT_TO_INT(DT_TO_UDINT(XDT) MOD 3600) / 60;
END_FUNCTION

FUNCTION MINUTE_TO_TIME : TIME
VAR_INPUT
	IN : REAL;
END_VAR

MINUTE_TO_TIME := DWORD_TO_TIME(REAL_TO_DWORD(IN * 60000.0));
END_FUNCTION

FUNCTION MONTH_BEGIN : DATE
VAR_INPUT
	idate : DATE;
END_VAR

MONTH_BEGIN := UDINT_TO_DATE(DATE_TO_UDINT(idate) - INT_TO_UDINT(DAY_OF_MONTH(idate) - 1) * 86400);
END_FUNCTION

FUNCTION MONTH_END : DATE
VAR_INPUT
	IDATE : DATE;
END_VAR

MONTH_END := UDINT_TO_DATE(DATE_TO_UDINT(SET_DATE(YEAR_OF_DATE(idate),MONTH_OF_DATE(idate)+1,1)) - 86400);
END_FUNCTION

FUNCTION MONTH_OF_DATE : INT
VAR_INPUT
	IDATE : DATE;
END_VAR

MONTH_OF_DATE := DAY_OF_YEAR(idate);
IF MONTH_OF_DATE < 32 THEN
	MONTH_OF_DATE := 1;
ELSIF LEAP_OF_DATE(IDATE) THEN
	MONTH_OF_DATE := (MONTH_OF_DATE * 53 + 1668) / 1623;
ELSE
	MONTH_OF_DATE := (MONTH_OF_DATE * 53 + 1700) / 1620;
END_IF;
END_FUNCTION

FUNCTION MULTIME : TIME
VAR_INPUT
	t : TIME;
	M : REAL;
END_VAR

MULTIME := DWORD_TO_TIME(REAL_TO_DWORD(DWORD_TO_REAL(TIME_TO_DWORD(t))*M));
END_FUNCTION

FUNCTION PERIOD : BOOL
VAR_INPUT
	d1 : DATE;
	dx : DATE;
	d2 : DATE;
END_VAR
VAR
	day1, day2, dayx : INT;
END_VAR

day1 := DAY_OF_YEAR(d1);
day2 := DAY_OF_YEAR(d2);
dayx := DAY_OF_YEAR(dx);
IF NOT LEAP_OF_DATE(dx) AND dayx > 58 THEN dayx := dayx + 1; END_IF;
IF NOT LEAP_OF_DATE(d1) AND day1 > 58 THEN day1 := day1 + 1; END_IF;
IF NOT LEAP_OF_DATE(d2) AND day2 > 58 THEN day2 := day2 + 1; END_IF;

IF day2 < day1 THEN
	(* the period spans over the new year *)
	PERIOD := dayx <= day2 OR dayx >= day1;
ELSE
	PERIOD := dayx >= day1 AND dayx <= day2;
END_IF;
END_FUNCTION

FUNCTION PERIOD2 : BOOL
VAR_INPUT
	DP : ARRAY[0..3,0..1] OF DATE;
	DX : DATE;
END_VAR

PERIOD2 := 	(DX >= DP[0,0] AND DX <= DP[0,1]) OR
			(DX >= DP[1,0] AND DX <= DP[1,1]) OR
			(DX >= DP[2,0] AND DX <= DP[2,1]) OR
			(DX >= DP[3,0] AND DX <= DP[3,1]);
END_FUNCTION

FUNCTION REFRACTION : REAL
VAR_INPUT
	ELEV : REAL;
END_VAR
VAR
	ELEV_work : REAL;
END_VAR
(* IEC 61131-3 does not let a POU assign to its inputs, so the body works on copies. *)
ELEV_work := ELEV;

ELEV_work := LIMIT(-1.9, ELEV_work, 80.0);
REFRACTION := 0.0174532925199433 / TAN(0.0174532925199433 * (ELEV_work + 10.3 / (ELEV_work + 5.11)));
END_FUNCTION

FUNCTION_BLOCK RTC_2
VAR_INPUT
	SET : BOOL;
	SDT : DT;
	SMS : INT;
	DEN : BOOL;
	OFS : INT;
END_VAR
VAR_OUTPUT
	UDT : DT;
	LOCAL_DT : DT;
	DSO : BOOL;
	XMS : INT;
END_VAR
VAR
	RT : RTC_MS;
END_VAR

(* call rtc *)
RT(SET := SET, SDT := SDT, SMS := SMS);
UDT := rt.xdt;
XMS := rt.XMS;

(* check for daylight savings time and set dso output *)
DSO := DST(udt) AND DEN;

(* calculate time offset and set ldt output *)
LOCAL_DT := UDINT_TO_DT(DT_TO_UDINT(UDT) + INT_TO_DINT(ofs + BOOL_TO_INT(DSO)*60) * 60);
END_FUNCTION_BLOCK

FUNCTION_BLOCK RTC_MS
VAR_INPUT
	SET : BOOL;
	SDT : DT;
	SMS : INT;
END_VAR
VAR_OUTPUT
	XDT : DT;
	XMS : INT;
END_VAR
VAR
	init: BOOL;
	last: DWORD;
	Tx: DWORD;
END_VAR

tx := T_PLC_MS();
IF set OR NOT init THEN
	(* clock needs to be set when set is true or after power up *)
	init := TRUE;
	xdt := SDT;
	XMS := SMS;
ELSE
	XMS := XMS + DWORD_TO_INT(ULINT_TO_DWORD((DWORD_TO_ULINT(tx) + 4294967296 - DWORD_TO_ULINT(last)) MOD 4294967296));
	(* check if one second has expired *)
	IF XMS > 999 THEN
		XDT := XDT + T#1s;
		XMS := XMS - 1000;
	END_IF;
END_IF;
last := tx;
END_FUNCTION_BLOCK

FUNCTION SDT_TO_DATE : DATE
VAR_INPUT
	DTI : SDT;
END_VAR

SDT_TO_DATE := SET_DATE(DTI.YEAR, DTI.MONTH, DTI.DAY);
END_FUNCTION

FUNCTION SDT_TO_DT : DT
VAR_INPUT
	DTI : SDT;
END_VAR

SDT_TO_DT := SET_DT(DTI.YEAR, DTI.MONTH, DTI.DAY, DTI.HOUR, DTI.MINUTE, DTI.SECOND);
END_FUNCTION

FUNCTION SDT_TO_TOD : TOD
VAR_INPUT
	DTI : SDT;
END_VAR

SDT_TO_TOD := UDINT_TO_TOD(INT_TO_UDINT(DTI.HOUR) * 3600000 + INT_TO_UDINT(DTI.MINUTE) * 60000 + INT_TO_UDINT(DTI.SECOND) * 1000 + INT_TO_UDINT(DTI.MS));
END_FUNCTION

FUNCTION SECOND : REAL
VAR_INPUT
	itod : TOD;
END_VAR

SECOND := UDINT_TO_REAL(TOD_TO_UDINT(itod) - TOD_TO_UDINT(itod)/60000 * 60000) / 1000.0;
END_FUNCTION

FUNCTION SECOND_OF_DT : INT
VAR_INPUT
	XDT : DT;
END_VAR

SECOND_OF_DT := UDINT_TO_INT(DT_TO_UDINT(XDT) MOD 60);
END_FUNCTION

FUNCTION SECOND_TO_TIME : TIME
VAR_INPUT
	IN : REAL;
END_VAR

SECOND_TO_TIME := DWORD_TO_TIME(REAL_TO_DWORD(IN * 1000.0));
END_FUNCTION

FUNCTION SET_DATE : DATE
VAR_INPUT
	YEAR : INT;
	MONTH : INT;
	DAY : INT;
END_VAR
VAR
	count : INT;
	ofs: ARRAY[1..12] OF INT := 0, 31, 59, 90, 120, 151, 181, 212, 243, 273, 304, 334;

	ENDIF: BOOL;
END_VAR

IF (MONTH > 2) AND (year MOD 4 = 0)
THEN (* we add one day for leap year *)
	SET_DATE := UDINT_TO_DATE((INT_TO_UDINT(ofs[MONTH] + day ) + (INT_TO_UDINT(year) * 1461 - 2878169) / 4)*86400);
ELSE
	SET_DATE := UDINT_TO_DATE((INT_TO_UDINT(ofs[MONTH] + day - 1 ) + (INT_TO_UDINT(year) * 1461 - 2878169) / 4)*86400);
END_IF;

// old code
// IF month > 2 THEN
// 	count := (month - 1) * 30;
// 	IF month > 7 THEN count := count + SHR(month - 3,1); ELSE count := count + SHR(month - 4,1); END_IF;
// 	(* chech for leap year and add one day if true *)
// 	IF year MOD 4 = 0 THEN count := count + 1; END_IF;
// ELSE
// 	count := (month - 1) * 31;
// END_IF;
//
// SET_DATE := UDINT_TO_DATE((INT_TO_UDINT(count + day - 1) + (INT_TO_UDINT(year) * 1461 - 2878169) / 4) * 86400);
END_FUNCTION

FUNCTION SET_DT : DT
VAR_INPUT
	year : INT;
	month : INT;
	day : INT;
	hour : INT;
	minute : INT;
	second : INT;
END_VAR

SET_DT := UDINT_TO_DT(DATE_TO_UDINT(SET_DATE(YEAR, MONTH, day)) + INT_TO_UDINT(SECOND) + INT_TO_UDINT(MINUTE) * 60 + INT_TO_UDINT(HOUR) * 3600);
END_FUNCTION

FUNCTION SET_TOD : TOD
VAR_INPUT
	hour : INT;
	minute : INT;
	second : REAL;
END_VAR

SET_TOD := UDINT_TO_TOD(REAL_TO_UDINT(SECOND * 1000.0) + INT_TO_UDINT(MINUTE) * 60000 + INT_TO_UDINT(HOUR) * 3600000);
END_FUNCTION

FUNCTION SUN_MIDDAY : TOD
VAR_INPUT
	LON : REAL;
	UTC : DATE;
END_VAR
VAR
	T : REAL;
	OFFSET : REAL;
END_VAR

T := INT_TO_REAL(DAY_OF_YEAR(utc));
OFFSET := -0.1752 * SIN(0.033430 * T + 0.5474) - 0.1340 * SIN(0.018234 * T - 0.1939);
SUN_MIDDAY := HOUR_TO_TOD(12.0 - OFFSET - lon * 0.0666666666666);
END_FUNCTION

FUNCTION_BLOCK SUN_POS
VAR_INPUT
	latitude : REAL;				(* latitude of geographical position  *)
	longitude : REAL;				(* longitude of geographical position  *)
	utc : DT;						(*	world time				*)
END_VAR
VAR_OUTPUT
	B: REAL;
	H : REAL;
	HR: REAL;
END_VAR
VAR_TEMP
	g: REAL;
	a: REAL;
	d: REAL;
	t1: REAL;
	n: REAL;
	e: REAL;
	c: REAL;
	tau: REAL;
	sin_d: REAL;
	rlat: REAL;
	sin_lat: REAL;
	cos_lat: REAL;
	cos_tau: REAL;
	cos_d: REAL;
END_VAR

(* n is the julian date and the number of days since 1.1.2000-12:00 midday *)
(* be careful for step7 date startes 1.1.1990 instead of 1.1.1970 *)
(* for step7 this line must change *)
n := UDINT_TO_REAL(DT_TO_UDINT(UTC) - 946728000) * 0.000011574074074074;
g :=MODR(6.240040768 + 0.01720197 * n, math.PI2);
d := MODR(4.89495042 + 0.017202792 * n, math.PI2) + 0.033423055 * SIN(g) + 0.000349066 * SIN(2.0*g);
e := 0.409087723 - 0.000000006981317008 * n;
cos_d := COS(d);
sin_d := SIN(d);
a := ATAN(COS(e) * sin_d / cos_d);
IF cos_d < 0.0 THEN a := a + math.PI; END_IF;
c := ASIN(SIN(e) * sin_d);

(* also here we must be very careful utc is from 1.1.1970 for step7 the formula must change *)
tau := RAD(MODR(6.697376 + (n - 0.25) * 0.0657098245037645 + DWORD_TO_REAL(TOD_TO_DWORD(DT_TO_TOD(utc))) * 0.0000002785383333, 24.0) * 15.0 + longitude) - a;
rlat := RAD(latitude);
sin_lat := SIN(rlat);
cos_lat := COS(rlat);
cos_tau := COS(tau);
t1 := cos_tau * sin_lat - TAN(c) * cos_lat;
B := ATAN(SIN(tau) / t1);
IF t1< 0.0 THEN B := B + math.PI2; ELSE B := B + math.PI; END_IF;
B := DEG(MODR(B, math.PI2));
h := DEG(ASIN(COS(C) * cos_tau * cos_lat +SIN(c) * sin_lat));
IF h > 180.0 THEN h := h - 360.0; END_IF;
(* consider refraction *)
HR := h + REFRACTION(h);
END_FUNCTION_BLOCK

FUNCTION_BLOCK SUN_TIME
VAR_INPUT
	LATITUDE : REAL;				(* latitude of geographical position  *)
	LONGITUDE : REAL;				(* longitude of geographical position  *)
	UTC : DATE;						(*	world time	*)
	H : REAL := -0.83333333333;	(* heighth above horizon for sunrise *)
END_VAR
VAR_OUTPUT
	MIDDAY : TOD;			(*	astrological midday in hours when sun stands at south direction	*)
	SUN_RISE : TOD;				(*	sun rise for current day in local time *)
	SUN_SET : TOD;				(*	sun set for current day in local time *)
	SUN_DECLINATION : REAL;		(*	sun declination above horizon at midday in degrees	*)
END_VAR
VAR
	dk: REAL;						(* sun declination at midday *)
	delta: TIME;					(* delta from midday for sunrise and sunset  *)
	b: REAL;
END_VAR

B := latitude * 0.0174532925199433;
MIDDAY := SUN_MIDDAY(longitude, utc);
DK := 0.40954 * SIN(0.0172 * (INT_TO_REAL(DAY_OF_YEAR(utc)) - 79.35));
sun_declination := DEG(DK);
IF sun_declination > 180.0 THEN sun_declination := sun_declination - 360.0; END_IF;
sun_declination := 90.0 - LATITUDE + sun_declination;
delta := HOUR_TO_TIME(ACOS((SIN(RAD(H)) - SIN(B) * SIN(DK)) / (COS(B) * COS(DK))) * 3.819718632);
sun_rise := MIDDAY - delta;
sun_set := MIDDAY + delta;
END_FUNCTION_BLOCK

FUNCTION TIMECHECK : BOOL
VAR_INPUT
	TD : TOD;
	START : TOD;
	STOP : TOD;
END_VAR

IF stop < start THEN
	TIMECHECK := start <= TD OR TD < stop;
ELSE
	TIMECHECK := start <= TD AND TD < stop;
END_IF;
END_FUNCTION

FUNCTION UTC_TO_LTIME : DT
VAR_INPUT
	UTC : DT;
	DST_ENABLE : BOOL;
	TIME_ZONE_OFFSET : INT;
END_VAR
VAR
	tmp: INT;
END_VAR

tmp := TIME_ZONE_OFFSET * 60 + BOOL_TO_INT(DST_ENABLE AND DST(UTC)) * 3600;
IF tmp < 0 THEN
	tmp := ABS(tmp);
	UTC_TO_LTIME := UDINT_TO_DT(DT_TO_UDINT(UTC) -  INT_TO_UDINT(tmp));
ELSE
	UTC_TO_LTIME := UDINT_TO_DT(DT_TO_UDINT(UTC) +  INT_TO_UDINT(tmp));
END_IF;
END_FUNCTION

FUNCTION WORK_WEEK : INT
VAR_INPUT
	idate : DATE;
END_VAR
VAR
	d1 : DATE;
	w1 : INT;
	ds: DWORD;
	yr: INT;
	w31: INT;
	w01: INT;
	wm: INT;
END_VAR

(* calculate january 1st of the year of idate. *)
yr := YEAR_OF_DATE(idate);
d1 := YEAR_BEGIN(yr);
(* weekday of d1 *)
w1 := DAY_OF_WEEK(d1);
(* offset of the monday of the last calendar week of the previous year *)
(* if the first day of the year is later than thursday, the last calendar week starts on the monday before *)
(* if the first day of the year is a thursday or earlier, the first calendar week starts 2 mondays before *)
IF w1 < 5 THEN
	ds := ULINT_TO_DWORD(DATE_TO_ULINT(d1) - INT_TO_ULINT(w1+6) * 86400);
ELSE
	ds := ULINT_TO_DWORD(DATE_TO_ULINT(d1) - INT_TO_ULINT(w1-1) * 86400);
END_IF;

(* calendar week of the input date *)
WORK_WEEK := ULINT_TO_INT((DATE_TO_ULINT(idate) - DWORD_TO_ULINT(ds)) / 604800);

(* correction if work_week = 0 *)
IF work_week = 0 THEN
	(* work_week needs to be 53 when 1.jan of the year before is thursday or dec 31. is thursday. *)
	(* first and last weekday of a year is equal and one more day for a leap_year. *)
	IF w1 > 1 THEN w31 := w1 - 1; ELSE W31 := 7; END_IF;
	IF LEAP_YEAR(yr - 1) AND w31 > 1 THEN w01 := W31 - 1; ELSE w1 := 7; END_IF;
	(* if first or last day of a year is a thursday, the year has 53 weeks *)
	WORK_WEEK := 52 + BOOL_TO_INT(w31 = 4 OR w01 = 4);
ELSE
	(* end of year calculation *)
	(* calculated the first and last weekday *)
	IF leap_year(yr) THEN
		IF w1 < 7 THEN w31 := w1 + 1; ELSE w31 := 1; END_IF;
	ELSE
		w31 := w1;
	END_IF;
	(* if first or last day is thursday then the year has 53 weeks otherwise only 52 *)
	wm := 52 + BOOL_TO_INT(w31 = 4 OR w1 = 4);
	IF WORK_WEEK > wm THEN WORK_WEEK := 1; END_IF;
END_IF;
END_FUNCTION

FUNCTION YEAR_BEGIN : DATE
VAR_INPUT
	y : INT;
END_VAR

YEAR_BEGIN := UDINT_TO_DATE((INT_TO_UDINT(y) * 1461 - 2878169) / 4 * 86400);
END_FUNCTION

FUNCTION YEAR_END : DATE
VAR_INPUT
	y : INT;
END_VAR

YEAR_END := UDINT_TO_DATE((INT_TO_UDINT(y) * 1461 - 2876712) / 4 * 86400);
END_FUNCTION

FUNCTION YEAR_OF_DATE : INT
VAR_INPUT
	IDATE : DATE;
END_VAR

YEAR_OF_DATE := UDINT_TO_INT((DATE_TO_UDINT(idate) + 43200) / 31557600 + 1970);
END_FUNCTION

TYPE CALENDAR :
STRUCT
	UTC : DT;					(* world time UTC *)
	LOCAL_DT : DT;					(* local time *)
	LOCAL_DATE : DATE;				(* local date *)
	LOCAL_TOD : TOD;					(* local time of day *)
	YEAR : INT;					(* year of LDATE *)
	MONTH : INT;				(* month of LDATE *)
	DAY : INT;					(* day of LDATE *)
	WEEKDAY : INT;				(* weekday of LDATE *)
	OFFSET : INT;				(* Time Zone Offset for Local time in minutes *)
	DST_EN : BOOL;				(* daylight savings time enable *)
	DST_ON : BOOL;				(* true when daylight savings time os on *)
	NAME : STRING(5);			(* name of time zone *)
	LANGUAGE : INT;			(* location number pls see location setup *)
	LONGITUDE : REAL;			(* longitude of current location *)
	LATITUDE : REAL;			(* latitude of current location *)
	SUN_RISE : TOD;				(* sun_rise for current location *)
	SUN_SET : TOD;				(* sun_set for current location *)
	SUN_MIDDAY : TOD;			(* worldtime when sun stands at south position *)
	SUN_HEIGTH : REAL	;		(* suns heigth at midday, south position *)
	SUN_HOR : REAL;			(* sun angle horizontal 0 = north in degrees *)
	SUN_VER : REAL;			(* sun angle vertical above horizon in degrees *)
	NIGHT : BOOL;				(* true between sun_set and sun_rise *)
	HOLIDAY : BOOL;			(* true when holiday *)
	HOLY_NAME : STRING(30);	(* name of holiday *)
	WORK_WEEK : INT;			(* current work week *)
END_STRUCT
END_TYPE

TYPE COMPLEX :
STRUCT
	re : REAL;
	im : REAL;
END_STRUCT
END_TYPE

TYPE CONSTANTS_LANGUAGE :
STRUCT
	(* Language Setup *)
	DEFAULT : INT := 1; (* 1=english, 2=german 3=french *)
	LMAX : INT := 3;
	WEEKDAYS : ARRAY[1..3, 1..7] OF STRING(10) :=	'Monday', 'Tuesday', 'Wednesday', 'Thursday', 'Friday', 'Saturday', 'Sunday',
													'Montag', 'Dienstag', 'Mittwoch', 'Donnerstag', 'Freitag', 'Samstag', 'Sonntag',
													'Lundi', 'Mardi', 'Mercredi', 'Jeudi', 'Vendredi', 'Samedi', 'Dimanche';
	WEEKDAYS2 : ARRAY[1..3, 1..7] OF STRING(2) :=	'Mo', 'Tu', 'We', 'Th', 'Fr', 'Sa', 'Su',
													'Mo', 'Di', 'Mi', 'Do', 'Fr', 'Sa', 'So',
													'Lu', 'Ma', 'Me', 'Je', 'Ve', 'Sa', 'Di';
	MONTHS : ARRAY[1..3, 1..12] OF STRING(10) :=	'January', 'February', 'March', 'April', 'May', 'June', 'July', 'August', 'September', 'October', 'November', 'December',
													'Januar', 'Februar', 'März', 'April', 'Mai', 'Juni', 'Juli', 'August', 'September', 'Oktober', 'November', 'Dezember',
													'Janvier', 'Février', 'mars', 'Avril', 'Mai', 'Juin', 'Juillet', 'Août', 'Septembre', 'Octobre', 'Novembre', 'Decembre';
	MONTHS3 : ARRAY[1..3, 1..12] OF STRING(3) :=	'Jan', 'Feb', 'Mar', 'Apr', 'May', 'Jun', 'Jul', 'Aug', 'Sep', 'Oct', 'Nov', 'Dec',
													'Jan', 'Feb', 'Mrz', 'Apr', 'Mai', 'Jun', 'Jul', 'Aug', 'Sep', 'Okt', 'Nov', 'Dez',
													'Jan', 'Fev', 'Mar', 'Avr', 'Mai', 'Jun', 'Jul', 'Aou', 'Sep', 'Oct', 'Nov', 'Dec';
	DIRS : ARRAY[1..3,0..15] OF STRING(3) :=		'N', 'NNE', 'NE', 'ENE', 'E', 'ESE', 'SE', 'SSE', 'S', 'SSW', 'SW', 'WSW', 'W', 'WNW', 'NW', 'NNW',
													'N', 'NNO', 'NO', 'ONO', 'O', 'OSO', 'SO', 'SSO', 'S', 'SSW', 'SW', 'WSW', 'W', 'WNW', 'NW', 'NNW',
													'N', 'NNO', 'NO', 'ONO', 'O', 'OSO', 'SO', 'SSO', 'S', 'SSW', 'SW', 'WSW', 'W', 'WNW', 'NW', 'NNW';
END_STRUCT
END_TYPE

TYPE CONSTANTS_LOCATION :
STRUCT
	(* location setup *)
	DEFAULT : INT := 1; (* 1=germany, 2=austria 3=france 4=belgium-german 5= italy-south tyrol *)
	LMAX : INT := 5;

	(* language spoken in the location *)
	LANGUAGE : ARRAY[1..5] OF INT := 2, 2, 3, 2, 2;

END_STRUCT
END_TYPE

TYPE CONSTANTS_MATH :
STRUCT
	PI : REAL := 	3.14159265358979323846264338327950288;		(* circle constant PI *)
	PI2 : REAL := 	6.28318530717958647692528676655900576;	(* PI * 2 *)
	PI4 : REAL :=  12.56637061435917295385057353311801152;	(* PI * 4 *)
	PI05 : REAL :=  1.5707963267949;							(* PI / 2 *)
	PI025 : REAL := 0.785398163397448;							(* PI / 4 *)
	PI_INV : REAL := 0.318309886183791;						(* 1 / PI *)
	E : REAL := 	2.71828182845904523536028747135266249;		(* Euler constant e *)
	E_INV : REAL := 0.367879441171442;							(* 1 / e *)
	SQ2 : REAL :=	1.4142135623731;							(* square root of 2 *)
	FACTS : ARRAY[0..12] OF DINT := 1,1,2,6,24,120,720,5040,40320,362880,3628800,39916800,479001600;
END_STRUCT
END_TYPE

TYPE CONSTANTS_PHYS :
STRUCT
	C : REAL := 299792458.0;				(* speed of light in m/s *)
	E : REAL := 1.60217653E-19;				(* elementary charge in coulomb = A * s *)
	G : REAL := 9.80665; 						(* gravitational acceleration in m / s² *)
	T0 : REAL := -273.15;						(* absolute zero in °C *)
	RU : REAL := 8.314472; 					(* universal gas constant in J / (mol · K) *)
	PN : REAL := 101325.0;					(* standard pressure in Pa *)
END_STRUCT
END_TYPE

TYPE CONSTANTS_SETUP :
STRUCT
	(* setup Parameters *)
	EXTENDED_ASCII : BOOL := TRUE;
	CHARNAMES : ARRAY[1..4] OF STRING(253) := ';"&quot;&&amp;<&lt;>&gt;&euro; &nbsp;¡&iexcl;¢&cent;£&pound;¤&curren;¥&yen;¦&brvbar;§&sect;¨&uml;©&copy;ª&ordf;«&laquo;¬&not;­&shy;®&reg;¯&macr;°&deg;±&plusmn;²&sup2;³&sup3;´&acute;µ&micro;¶&para;·&middot;¸&cedil;¹&sup1;º&ordm;»&raquo;¼&frac14;Û&Ucirc;',
		';¾&frac34;¿&iquest;À&Agrave;Á&Aacute;Â&Acirc;Ã&Atilde;Ä&Auml;Å&Aring;Æ&AElig;Ç&Ccedil;È&Egrave;É&Eacute;Ê&Ecirc;Ë&Euml;Ì&Igrave;Í&Iacute;Î&Icirc;Ï&Iuml;Ð&ETH;Ñ&Ntilde;Ò&Ograve;Ó&Oacute;Ô&Ocirc;Õ&Otilde;Ö&Ouml;×&times;Ø&Oslash;Ù&Ugrave;Ú&Uacute;½&frac12;',
		';Ü&Uuml;Ý&Yacute;Þ&THORN;ß&szlig;à&agrave;á&aacute;â&acirc;ã&atilde;ä&auml;å&aring;æ&aelig;ç&ccedil;è&egrave;é&eacute;ê&ecirc;ë&euml;ì&igrave;í&iacute;î&icirc;ï&iuml;ð&eth;ñ&ntilde;ò&ograve;ó&oacute;ô&ocirc;õ&otilde;ö&ouml;÷&divide;ø&oslash;ù&ugrave;',
		';ú&uacute;û&ucirc;ü&uuml;ý&yacute;þ&thorn;ÿ&yuml;';
	MTH_OFS : ARRAY[1..12] OF INT := 0,31,59,90,120,151,181,212,243,273,304,334;
	DECADES : ARRAY[0..8] OF REAL := 1.0,10.0,100.0,1000.0,10000.0,100000.0,1000000.0,10000000.0,100000000.0;
END_STRUCT
END_TYPE

TYPE ESR_DATA :
STRUCT
	TYP : BYTE;
	ADRESS : STRING(10);
	DS : DT;
	TS : TIME;
	DATA : ARRAY[0..7] OF BYTE;
END_STRUCT
END_TYPE

TYPE FRACTION :
STRUCT
	NUMERATOR : INT;
	DENOMINATOR : INT;
END_STRUCT
END_TYPE

TYPE HOLIDAY_DATA :
STRUCT
	NAME : STRING(30);
	DAY : SINT;
	MONTH : SINT;
	USE : SINT;
END_STRUCT
END_TYPE

TYPE REAL2 :
STRUCT
	R1 : REAL;	(* small value *)
	RX : REAL;	(* big value *)
END_STRUCT
END_TYPE

TYPE SDT :
STRUCT
	YEAR : INT;
	MONTH : INT;
	DAY : INT;
	WEEKDAY : INT;
	HOUR : INT;
	MINUTE : INT;
	SECOND : INT;
	MS : INT;
END_STRUCT
END_TYPE

TYPE TIMER_EVENT :
STRUCT
	TYP : BYTE;
	CHANNEL : BYTE;
	DAY : BYTE;
	START : TOD;
	DURATION : TIME;
	LAND : BYTE;
	LOR : BYTE;
	LAST : DT;
END_STRUCT
END_TYPE

TYPE VECTOR_3 :
STRUCT
	X : REAL;
	Y : REAL;
	Z : REAL;
END_STRUCT
END_TYPE

VAR_GLOBAL CONSTANT
	STRING_LENGTH : INT := 250;
	LIST_LENGTH : INT := 250;
END_VAR

VAR_GLOBAL
	MATH : CONSTANTS_MATH;
	PHYS : CONSTANTS_PHYS;
	LANGUAGE : CONSTANTS_LANGUAGE;
	SETUP : CONSTANTS_SETUP;
	LOCATION : CONSTANTS_LOCATION;
END_VAR

VAR_GLOBAL RETAIN

END_VAR
